C09105=1126.516,313.424,-77.649,-177.752,10.579,149.528
C09106=1126.520,313.176,-77.616,-177.755,10.576,149.528
C09107=1126.524,312.928,-77.584,-177.758,10.574,149.528
C09108=1126.528,312.680,-77.551,-177.761,10.571,149.528
C09109=1126.531,312.433,-77.519,-177.764,10.568,149.528
C09110=1126.536,312.184,-77.486,-177.767,10.567,149.529
C09111=1126.540,311.937,-77.453,-177.770,10.564,149.529
C09112=1126.544,311.688,-77.421,-177.773,10.562,149.529
C09113=1126.548,311.441,-77.389,-177.776,10.559,149.529
C09114=1126.552,311.193,-77.357,-177.779,10.556,149.529
C09115=1126.556,310.946,-77.324,-177.783,10.554,149.529
C09116=1126.560,310.698,-77.292,-177.786,10.551,149.530
C09117=1126.564,310.449,-77.259,-177.789,10.549,149.530
C09118=1126.568,310.202,-77.227,-177.792,10.546,149.530
C09119=1126.572,309.954,-77.194,-177.795,10.543,149.530
C09120=1126.577,309.706,-77.163,-177.798,10.541,149.530
C09121=1126.581,309.458,-77.130,-177.801,10.538,149.530
C09122=1126.584,309.210,-77.098,-177.805,10.536,149.531
C09123=1126.589,308.962,-77.065,-177.808,10.533,149.531
C09124=1126.592,308.715,-77.033,-177.811,10.531,149.531
C09125=1126.597,308.502,-77.005,-177.813,10.529,149.531
C09126=1126.600,308.289,-76.978,-177.816,10.527,149.531
C09127=1126.603,308.075,-76.950,-177.819,10.524,149.532
C09128=1126.607,307.862,-76.922,-177.821,10.522,149.532
C09129=1126.610,307.649,-76.895,-177.824,10.520,149.532
C09130=1126.614,307.436,-76.868,-177.827,10.518,149.532
C09131=1126.618,307.222,-76.840,-177.829,10.516,149.532
C09132=1126.621,307.009,-76.812,-177.832,10.513,149.532
C09133=1126.625,306.762,-76.779,-177.835,10.511,149.532
C09134=1126.629,306.514,-76.747,-177.838,10.509,149.533
C09135=1126.633,306.266,-76.715,-177.841,10.506,149.533
C09136=1126.637,306.017,-76.683,-177.844,10.504,149.533
C09137=1126.642,305.770,-76.652,-177.847,10.501,149.533
C09138=1126.645,305.522,-76.620,-177.851,10.499,149.533
C09139=1126.650,305.274,-76.587,-177.854,10.496,149.533
C09140=1126.653,305.026,-76.555,-177.857,10.493,149.534
C09141=1126.658,304.778,-76.524,-177.860,10.491,149.534
C09142=1126.662,304.530,-76.492,-177.863,10.488,149.534
C09143=1126.666,304.282,-76.460,-177.866,10.485,149.534
C09144=1126.670,304.035,-76.428,-177.869,10.483,149.534
C09145=1126.675,303.786,-76.396,-177.873,10.480,149.535
C09146=1126.678,303.538,-76.364,-177.876,10.478,149.535
C09147=1126.683,303.291,-76.332,-177.878,10.476,149.535
C09148=1126.687,303.043,-76.300,-177.881,10.473,149.535
C09149=1126.691,302.795,-76.268,-177.885,10.471,149.535
C09150=1126.695,302.547,-76.237,-177.888,10.468,149.536
C09151=1126.699,302.299,-76.205,-177.891,10.466,149.536
C09152=1126.703,302.051,-76.172,-177.894,10.463,149.536
C09153=1126.708,301.803,-76.141,-177.897,10.460,149.536
C09154=1126.711,301.555,-76.109,-177.900,10.458,149.536
C09155=1126.715,301.307,-76.077,-177.904,10.455,149.536
C09156=1126.720,301.059,-76.046,-177.906,10.452,149.537
C09157=1126.724,300.811,-76.014,-177.910,10.450,149.537
C09158=1126.728,300.563,-75.982,-177.913,10.447,149.537
C09159=1126.732,300.316,-75.951,-177.915,10.446,149.537
C09160=1126.736,300.068,-75.919,-177.918,10.443,149.537
C09161=1126.740,299.820,-75.888,-177.922,10.440,149.538
C09162=1126.745,299.571,-75.856,-177.925,10.438,149.538
C09163=1126.749,299.323,-75.824,-177.928,10.435,149.538
C09164=1126.753,299.076,-75.792,-177.931,10.432,149.538
C09165=1126.757,298.827,-75.761,-177.934,10.430,149.538
C09166=1126.761,298.579,-75.729,-177.937,10.427,149.538
C09167=1126.765,298.332,-75.698,-177.941,10.425,149.539
C09168=1126.769,298.084,-75.666,-177.943,10.422,149.539
C09169=1126.773,297.836,-75.635,-177.947,10.420,149.539
C09170=1126.777,297.588,-75.603,-177.950,10.417,149.539
C09171=1126.781,297.340,-75.573,-177.953,10.414,149.539
C09172=1126.785,297.092,-75.541,-177.955,10.412,149.539
C09173=1126.789,296.845,-75.509,-177.959,10.410,149.540
C09174=1126.794,296.596,-75.478,-177.962,10.407,149.540
C09175=1126.798,296.348,-75.446,-177.965,10.405,149.540
C09176=1126.803,296.100,-75.415,-177.968,10.402,149.540
C09177=1126.806,295.852,-75.383,-177.971,10.400,149.540
C09178=1126.811,295.604,-75.352,-177.974,10.397,149.540
C09179=1126.815,295.356,-75.321,-177.977,10.394,149.541
C09180=1126.818,295.109,-75.290,-177.980,10.392,149.541
C09181=1126.822,294.895,-75.263,-177.983,10.390,149.541
C09182=1126.826,294.682,-75.236,-177.985,10.388,149.541
C09183=1126.829,294.468,-75.209,-177.988,10.385,149.541
C09184=1126.833,294.255,-75.182,-177.991,10.383,149.541
C09185=1126.836,294.042,-75.155,-177.994,10.381,149.542
C09186=1126.840,293.828,-75.129,-177.996,10.379,149.542
C09187=1126.843,293.615,-75.101,-177.999,10.377,149.542
C09188=1126.847,293.401,-75.074,-178.002,10.374,149.542
C09189=1126.851,293.153,-75.044,-178.005,10.372,149.542
C09190=1126.855,292.905,-75.012,-178.008,10.369,149.543
C09191=1126.859,292.657,-74.981,-178.011,10.367,149.543
C09192=1126.864,292.409,-74.950,-178.013,10.365,149.543
C09193=1126.867,292.162,-74.919,-178.017,10.362,149.543
C09194=1126.872,291.914,-74.888,-178.020,10.359,149.543
C09195=1126.876,291.665,-74.857,-178.023,10.357,149.543
C09196=1126.880,291.418,-74.826,-178.026,10.354,149.544
C09197=1126.884,291.169,-74.795,-178.029,10.352,149.544
C09198=1126.889,290.921,-74.764,-178.032,10.349,149.544
C09199=1126.892,290.673,-74.733,-178.036,10.347,149.544
C09200=1126.896,290.426,-74.702,-178.039,10.344,149.544
C09201=1126.901,290.178,-74.671,-178.042,10.341,149.545
C09202=1126.905,289.929,-74.640,-178.044,10.339,149.545
C09203=1126.909,289.681,-74.609,-178.048,10.337,149.545
C09204=1126.912,289.433,-74.578,-178.050,10.334,149.545
C09205=1126.917,289.185,-74.547,-178.053,10.331,149.545
C09206=1126.922,288.937,-74.516,-178.057,10.329,149.545
C09207=1126.926,288.689,-74.485,-178.060,10.326,149.545
C09208=1126.929,288.441,-74.455,-178.063,10.324,149.546
C09209=1126.934,288.193,-74.424,-178.066,10.321,149.546
C09210=1126.938,287.945,-74.392,-178.069,10.319,149.546
C09211=1126.942,287.697,-74.362,-178.072,10.316,149.546
C09212=1126.946,287.449,-74.331,-178.075,10.314,149.546
C09213=1126.950,287.201,-74.300,-178.078,10.311,149.547
C09214=1126.955,286.953,-74.270,-178.081,10.309,149.547
C09215=1126.958,286.704,-74.239,-178.084,10.306,149.547
C09216=1126.963,286.456,-74.208,-178.087,10.304,149.547
C09217=1126.967,286.209,-74.178,-178.090,10.301,149.547
C09218=1126.971,285.960,-74.147,-178.093,10.298,149.547
C09219=1126.975,285.712,-74.116,-178.097,10.296,149.548
C09220=1126.980,285.464,-74.085,-178.100,10.293,149.548
C09221=1126.984,285.217,-74.055,-178.103,10.291,149.548
C09222=1126.988,284.968,-74.024,-178.105,10.289,149.548
C09223=1126.992,284.720,-73.993,-178.108,10.286,149.548
C09224=1126.996,284.472,-73.963,-178.112,10.284,149.549
C09225=1127.001,284.223,-73.933,-178.115,10.281,149.549
C09226=1127.004,283.975,-73.903,-178.118,10.278,149.549
C09227=1127.009,283.727,-73.872,-178.121,10.276,149.549
C09228=1127.013,283.480,-73.842,-178.124,10.273,149.549
C09229=1127.017,283.231,-73.811,-178.127,10.270,149.549
C09230=1127.022,282.983,-73.780,-178.130,10.268,149.549
C09231=1127.025,282.736,-73.750,-178.133,10.265,149.550
C09232=1127.030,282.487,-73.720,-178.136,10.263,149.550
C09233=1127.034,282.239,-73.689,-178.139,10.261,149.550
C09234=1127.038,281.991,-73.658,-178.142,10.258,149.550
C09235=1127.042,281.743,-73.628,-178.145,10.255,149.550
C09236=1127.047,281.494,-73.598,-178.148,10.253,149.551
C09237=1127.050,281.281,-73.572,-178.151,10.250,149.551
C09238=1127.054,281.068,-73.545,-178.154,10.248,149.551
C09239=1127.058,280.854,-73.520,-178.157,10.246,149.551
C09240=1127.061,280.641,-73.494,-178.160,10.243,149.551
C09241=1127.065,280.427,-73.468,-178.163,10.241,149.552
C09242=1127.068,280.214,-73.442,-178.166,10.238,149.552
C09243=1127.072,280.001,-73.415,-178.169,10.236,149.552
C09244=1127.075,279.787,-73.390,-178.172,10.234,149.552
C09245=1127.080,279.539,-73.359,-178.176,10.230,149.552
C09246=1127.084,279.291,-73.329,-178.179,10.228,149.553
C09247=1127.089,279.043,-73.299,-178.182,10.225,149.553
C09248=1127.093,278.795,-73.268,-178.185,10.223,149.553
C09249=1127.097,278.547,-73.239,-178.189,10.219,149.553
C09250=1127.101,278.298,-73.208,-178.192,10.217,149.553
C09251=1127.105,278.050,-73.178,-178.195,10.214,149.553
C09252=1127.109,277.802,-73.148,-178.198,10.212,149.554
C09253=1127.114,277.554,-73.118,-178.202,10.208,149.554
C09254=1127.118,277.306,-73.088,-178.205,10.206,149.554
C09255=1127.122,277.058,-73.059,-178.208,10.203,149.554
C09256=1127.126,276.810,-73.028,-178.211,10.200,149.554
C09257=1127.130,276.561,-72.998,-178.215,10.198,149.555
C09258=1127.134,276.313,-72.968,-178.218,10.194,149.555
C09259=1127.138,276.065,-72.938,-178.222,10.192,149.555
C09260=1127.143,275.816,-72.908,-178.224,10.189,149.555
C09261=1127.147,275.569,-72.878,-178.227,10.186,149.555
C09262=1127.151,275.320,-72.849,-178.230,10.183,149.555
C09263=1127.155,275.072,-72.819,-178.234,10.181,149.556
C09264=1127.160,274.824,-72.788,-178.237,10.178,149.556
C09265=1127.164,274.576,-72.759,-178.240,10.176,149.556
C09266=1127.168,274.328,-72.730,-178.243,10.173,149.556
C09267=1127.172,274.080,-72.699,-178.246,10.170,149.556
C09268=1127.177,273.831,-72.669,-178.249,10.168,149.556
C09269=1127.181,273.583,-72.640,-178.252,10.165,149.556
C09270=1127.185,273.335,-72.610,-178.255,10.162,149.556
C09271=1127.189,273.087,-72.580,-178.258,10.159,149.557
C09272=1127.193,272.839,-72.551,-178.261,10.157,149.557
C09273=1127.198,272.591,-72.521,-178.263,10.154,149.557
C09274=1127.202,272.342,-72.491,-178.267,10.151,149.557
C09275=1127.206,272.094,-72.461,-178.270,10.149,149.557
C09276=1127.210,271.846,-72.432,-178.273,10.146,149.557
C09277=1127.215,271.598,-72.402,-178.276,10.143,149.557
C09278=1127.219,271.350,-72.373,-178.278,10.141,149.557
C09279=1127.223,271.101,-72.343,-178.281,10.138,149.558
C09280=1127.227,270.853,-72.314,-178.284,10.136,149.558
C09281=1127.231,270.605,-72.284,-178.287,10.133,149.558
C09282=1127.235,270.357,-72.254,-178.290,10.130,149.558
C09283=1127.239,270.109,-72.225,-178.292,10.128,149.558
C09284=1127.244,269.860,-72.195,-178.295,10.125,149.558
C09285=1127.249,269.612,-72.165,-178.298,10.123,149.558
C09286=1127.253,269.364,-72.136,-178.300,10.121,149.558
C09287=1127.257,269.115,-72.106,-178.303,10.118,149.558
C09288=1127.261,268.867,-72.077,-178.306,10.115,149.558
C09289=1127.265,268.619,-72.047,-178.308,10.113,149.559
C09290=1127.269,268.371,-72.018,-178.311,10.110,149.559
C09291=1127.274,268.122,-71.989,-178.314,10.108,149.559
C09292=1127.278,267.874,-71.959,-178.317,10.106,149.559
C09293=1127.281,267.661,-71.934,-178.318,10.103,149.559
C09294=1127.285,267.447,-71.909,-178.321,10.101,149.559
C09295=1127.289,267.234,-71.884,-178.324,10.099,149.559
C09296=1127.292,267.020,-71.858,-178.326,10.097,149.559
C09297=1127.297,266.806,-71.833,-178.328,10.094,149.559
C09298=1127.300,266.593,-71.808,-178.330,10.092,149.559
C09299=1127.304,266.379,-71.783,-178.333,10.090,149.559
C09300=1127.307,266.166,-71.758,-178.335,10.088,149.560
C09301=1127.312,265.918,-71.728,-178.337,10.086,149.560
C09302=1127.316,265.669,-71.699,-178.339,10.084,149.560
C09303=1127.320,265.421,-71.669,-178.342,10.081,149.560
C09304=1127.324,265.173,-71.640,-178.344,10.079,149.560
C09305=1127.329,264.924,-71.611,-178.347,10.077,149.560
C09306=1127.333,264.676,-71.582,-178.350,10.075,149.560
C09307=1127.338,264.428,-71.553,-178.352,10.072,149.560
C09308=1127.341,264.180,-71.524,-178.356,10.069,149.560
C09309=1127.345,263.932,-71.494,-178.360,10.066,149.561
C09310=1127.350,263.683,-71.466,-178.363,10.063,149.561
C09311=1127.354,263.435,-71.436,-178.367,10.059,149.561
C09312=1127.359,263.187,-71.407,-178.371,10.056,149.561
C09313=1127.363,262.938,-71.378,-178.374,10.054,149.562
C09314=1127.367,262.690,-71.349,-178.378,10.050,149.562
C09315=1127.371,262.442,-71.320,-178.382,10.047,149.562
C09316=1127.375,262.193,-71.291,-178.385,10.044,149.562
C09317=1127.380,261.946,-71.262,-178.389,10.041,149.562
C09318=1127.384,261.697,-71.233,-178.392,10.038,149.563
C09319=1127.389,261.448,-71.204,-178.396,10.035,149.563
C09320=1127.392,261.200,-71.175,-178.400,10.032,149.563
C09321=1127.397,260.952,-71.146,-178.403,10.029,149.563
C09322=1127.401,260.704,-71.117,-178.406,10.025,149.563
C09323=1127.405,260.456,-71.089,-178.410,10.023,149.563
C09324=1127.409,260.207,-71.060,-178.413,10.020,149.564
C09325=1127.414,259.960,-71.031,-178.416,10.017,149.564
C09326=1127.419,259.711,-71.002,-178.419,10.014,149.564
C09327=1127.422,259.463,-70.973,-178.423,10.011,149.564
C09328=1127.427,259.214,-70.944,-178.426,10.008,149.564
C09329=1127.432,258.966,-70.916,-178.429,10.005,149.564
C09330=1127.435,258.718,-70.887,-178.433,10.002,149.564
C09331=1127.440,258.469,-70.858,-178.435,9.999,149.564
C09332=1127.444,258.221,-70.829,-178.438,9.996,149.565
C09333=1127.448,257.973,-70.801,-178.441,9.994,149.565
C09334=1127.453,257.724,-70.772,-178.444,9.991,149.565
C09335=1127.456,257.476,-70.744,-178.448,9.987,149.565
C09336=1127.461,257.228,-70.715,-178.451,9.985,149.565
C09337=1127.466,256.979,-70.686,-178.454,9.982,149.565
C09338=1127.470,256.731,-70.658,-178.456,9.979,149.565
C09339=1127.474,256.483,-70.629,-178.459,9.976,149.565
C09340=1127.478,256.234,-70.601,-178.462,9.973,149.565
C09341=1127.483,255.986,-70.572,-178.465,9.970,149.565
C09342=1127.486,255.738,-70.544,-178.465,9.969,149.565
C09343=1127.491,255.489,-70.515,-178.464,9.969,149.565
C09344=1127.496,255.241,-70.487,-178.465,9.967,149.565
C09345=1127.499,254.993,-70.458,-178.464,9.966,149.564
C09346=1127.504,254.744,-70.429,-178.465,9.965,149.564
C09347=1127.508,254.496,-70.401,-178.465,9.964,149.564
C09348=1127.513,254.247,-70.373,-178.466,9.963,149.564
C09349=1127.516,254.034,-70.347,-178.467,9.961,149.564
C09350=1127.519,253.820,-70.324,-178.468,9.960,149.564
C09351=1127.523,253.606,-70.299,-178.470,9.959,149.564
C09352=1127.528,253.393,-70.274,-178.471,9.957,149.564
C09353=1127.531,253.179,-70.250,-178.472,9.955,149.564
C09354=1127.535,252.965,-70.226,-178.474,9.954,149.564
C09355=1127.538,252.752,-70.201,-178.476,9.952,149.564
C09356=1127.542,252.538,-70.176,-178.478,9.950,149.564
C09357=1127.546,252.290,-70.149,-178.480,9.948,149.564
C09358=1127.551,252.041,-70.120,-178.484,9.946,149.564
C09359=1127.555,251.793,-70.092,-178.487,9.943,149.564
C09360=1127.559,251.545,-70.063,-178.490,9.940,149.565
C09361=1127.563,251.297,-70.034,-178.494,9.937,149.565
C09362=1127.568,251.048,-70.006,-178.498,9.934,149.565
C09363=1127.572,250.800,-69.978,-178.502,9.931,149.565
C09364=1127.576,250.551,-69.949,-178.506,9.928,149.566
C09365=1127.581,250.303,-69.921,-178.510,9.925,149.566
C09366=1127.584,250.054,-69.893,-178.515,9.921,149.566
C09367=1127.590,249.806,-69.865,-178.520,9.917,149.567
C09368=1127.593,249.558,-69.837,-178.525,9.913,149.567
C09369=1127.598,249.309,-69.808,-178.530,9.909,149.568
C09370=1127.602,249.061,-69.780,-178.536,9.904,149.568
C09371=1127.607,248.813,-69.752,-178.541,9.900,149.569
C09372=1127.611,248.564,-69.724,-178.548,9.895,149.569
C09373=1127.615,248.316,-69.696,-178.554,9.891,149.570
C09374=1127.619,248.068,-69.668,-178.560,9.886,149.570
C09375=1127.624,247.819,-69.641,-178.567,9.880,149.571
C09376=1127.628,247.570,-69.612,-178.574,9.875,149.571
C09377=1127.633,247.322,-69.584,-178.578,9.871,149.571
C09378=1127.637,247.075,-69.556,-178.580,9.868,149.571
C09379=1127.641,246.825,-69.529,-178.581,9.866,149.571
C09380=1127.646,246.577,-69.501,-178.583,9.864,149.571
C09381=1127.650,246.329,-69.472,-178.583,9.862,149.571
C09382=1127.655,246.080,-69.445,-178.585,9.860,149.571
C09383=1127.658,245.832,-69.417,-178.586,9.858,149.570
C09384=1127.663,245.584,-69.390,-178.588,9.856,149.570
C09385=1127.667,245.336,-69.362,-178.590,9.853,149.570
C09386=1127.672,245.086,-69.334,-178.591,9.851,149.570
C09387=1127.676,244.838,-69.306,-178.593,9.849,149.570
C09388=1127.680,244.590,-69.278,-178.595,9.847,149.570
C09389=1127.685,244.341,-69.251,-178.596,9.845,149.570
C09390=1127.689,244.093,-69.223,-178.598,9.843,149.570
C09391=1127.693,243.844,-69.196,-178.600,9.840,149.570
C09392=1127.698,243.596,-69.167,-178.602,9.838,149.570
C09393=1127.702,243.347,-69.139,-178.603,9.836,149.570
C09394=1127.706,243.099,-69.112,-178.605,9.833,149.570
C09395=1127.711,242.851,-69.084,-178.607,9.831,149.569
C09396=1127.715,242.603,-69.056,-178.609,9.829,149.569
C09397=1127.719,242.354,-69.029,-178.611,9.826,149.569
C09398=1127.724,242.106,-69.001,-178.613,9.824,149.569
C09399=1127.728,241.857,-68.974,-178.615,9.822,149.569
C09400=1127.732,241.609,-68.946,-178.617,9.820,149.569
C09401=1127.737,241.361,-68.919,-178.619,9.818,149.569
C09402=1127.741,241.112,-68.890,-178.621,9.815,149.569
C09403=1127.746,240.863,-68.863,-178.623,9.813,149.569
C09404=1127.750,240.615,-68.835,-178.626,9.810,149.569
C09405=1127.754,240.401,-68.812,-178.628,9.808,149.569
C09406=1127.757,240.187,-68.788,-178.629,9.807,149.569
C09407=1127.761,239.974,-68.764,-178.631,9.804,149.569
C09408=1127.765,239.760,-68.741,-178.634,9.802,149.570
C09409=1127.768,239.546,-68.717,-178.635,9.800,149.569
C09410=1127.772,239.332,-68.693,-178.638,9.798,149.570
C09411=1127.776,239.118,-68.670,-178.640,9.796,149.570
C09412=1127.780,238.905,-68.646,-178.642,9.794,149.570
C09413=1127.784,238.656,-68.618,-178.645,9.791,149.570
C09414=1127.788,238.408,-68.591,-178.647,9.789,149.570
C09415=1127.793,238.159,-68.564,-178.650,9.786,149.570
C09416=1127.797,237.910,-68.536,-178.652,9.784,149.570
C09417=1127.802,237.662,-68.508,-178.655,9.781,149.570
C09418=1127.806,237.414,-68.481,-178.658,9.778,149.570
C09419=1127.810,237.165,-68.455,-178.660,9.776,149.570
C09420=1127.814,236.917,-68.427,-178.663,9.773,149.570
C09421=1127.819,236.668,-68.400,-178.666,9.771,149.570
C09422=1127.823,236.420,-68.373,-178.669,9.768,149.571
C09423=1127.828,236.172,-68.345,-178.672,9.765,149.571
C09424=1127.832,235.923,-68.317,-178.675,9.762,149.571
C09425=1127.836,235.674,-68.290,-178.677,9.759,149.571
C09426=1127.841,235.426,-68.263,-178.680,9.756,149.571
C09427=1127.845,235.178,-68.235,-178.683,9.754,149.571
C09428=1127.849,234.929,-68.208,-178.686,9.751,149.571
C09429=1127.853,234.681,-68.182,-178.689,9.748,149.571
C09430=1127.858,234.432,-68.155,-178.692,9.745,149.571
C09431=1127.863,234.184,-68.127,-178.695,9.743,149.572
C09432=1127.867,233.936,-68.100,-178.698,9.740,149.572
C09433=1127.871,233.687,-68.072,-178.702,9.737,149.572
C09434=1127.876,233.438,-68.045,-178.705,9.734,149.572
C09435=1127.880,233.190,-68.019,-178.708,9.731,149.572
C09436=1127.884,232.941,-67.992,-178.711,9.728,149.572
C09437=1127.889,232.693,-67.965,-178.714,9.725,149.572
C09438=1127.893,232.444,-67.938,-178.718,9.722,149.573
C09439=1127.898,232.195,-67.910,-178.721,9.719,149.573
C09440=1127.901,231.947,-67.884,-178.724,9.715,149.573
C09441=1127.906,231.698,-67.857,-178.728,9.713,149.573
C09442=1127.911,231.450,-67.830,-178.731,9.709,149.573
C09443=1127.915,231.201,-67.802,-178.735,9.706,149.573
C09444=1127.919,230.953,-67.776,-178.738,9.703,149.573
C09445=1127.924,230.705,-67.749,-178.741,9.700,149.574
C09446=1127.929,230.456,-67.722,-178.745,9.696,149.574
C09447=1127.932,230.207,-67.695,-178.749,9.693,149.574
C09448=1127.937,229.959,-67.668,-178.753,9.689,149.574
C09449=1127.941,229.710,-67.641,-178.756,9.686,149.574
C09450=1127.945,229.462,-67.614,-178.760,9.682,149.574
C09451=1127.950,229.214,-67.587,-178.763,9.679,149.574
C09452=1127.955,228.965,-67.561,-178.767,9.676,149.575
C09453=1127.959,228.716,-67.535,-178.771,9.672,149.575
C09454=1127.963,228.468,-67.508,-178.774,9.669,149.575
C09455=1127.967,228.220,-67.481,-178.777,9.666,149.575
C09456=1127.972,227.971,-67.454,-178.781,9.662,149.575
C09457=1127.977,227.722,-67.428,-178.784,9.658,149.575
C09458=1127.981,227.474,-67.401,-178.788,9.655,149.575
C09459=1127.986,227.225,-67.374,-178.791,9.651,149.575
C09460=1127.990,226.977,-67.348,-178.794,9.649,149.576
C09461=1127.993,226.762,-67.325,-178.797,9.646,149.575
C09462=1127.997,226.549,-67.302,-178.800,9.642,149.576
C09463=1128.001,226.335,-67.280,-178.803,9.639,149.576
C09464=1128.005,226.121,-67.256,-178.806,9.636,149.576
C09465=1128.009,225.907,-67.234,-178.809,9.633,149.576
C09466=1128.012,225.693,-67.211,-178.811,9.630,149.576
C09467=1128.016,225.479,-67.188,-178.814,9.628,149.576
C09468=1128.020,225.265,-67.165,-178.816,9.625,149.576
C09469=1128.025,225.017,-67.139,-178.820,9.622,149.576
C09470=1128.029,224.768,-67.112,-178.823,9.618,149.576
C09471=1128.033,224.519,-67.086,-178.826,9.615,149.576
C09472=1128.037,224.271,-67.060,-178.828,9.612,149.576
C09473=1128.042,224.022,-67.034,-178.832,9.608,149.576
C09474=1128.046,223.774,-67.007,-178.834,9.605,149.576
C09475=1128.051,223.525,-66.981,-178.838,9.601,149.576
C09476=1128.055,223.276,-66.954,-178.840,9.598,149.576
C09477=1128.059,223.028,-66.929,-178.843,9.595,149.576
C09478=1128.064,222.779,-66.901,-178.846,9.592,149.576
C09479=1128.069,222.531,-66.876,-178.849,9.589,149.576
C09480=1128.073,222.283,-66.849,-178.851,9.586,149.576
C09481=1128.078,222.034,-66.823,-178.855,9.582,149.576
C09482=1128.082,221.785,-66.798,-178.857,9.579,149.576
C09483=1128.087,221.536,-66.770,-178.860,9.575,149.576
C09484=1128.091,221.288,-66.745,-178.862,9.572,149.576
C09485=1128.095,221.039,-66.718,-178.865,9.569,149.575
C09486=1128.099,220.791,-66.692,-178.867,9.566,149.575
C09487=1128.104,220.542,-66.667,-178.870,9.563,149.575
C09488=1128.108,220.294,-66.640,-178.872,9.560,149.575
C09489=1128.113,220.045,-66.614,-178.875,9.557,149.575
C09490=1128.118,219.796,-66.588,-178.877,9.554,149.575
C09491=1128.122,219.547,-66.562,-178.880,9.551,149.575
C09492=1128.126,219.299,-66.536,-178.882,9.547,149.575
C09493=1128.131,219.051,-66.510,-178.885,9.544,149.575
C09494=1128.136,218.802,-66.484,-178.887,9.541,149.575
C09495=1128.140,218.553,-66.458,-178.889,9.538,149.575
C09496=1128.144,218.305,-66.432,-178.892,9.535,149.575
C09497=1128.148,218.056,-66.406,-178.894,9.532,149.575
C09498=1128.152,217.807,-66.380,-178.896,9.529,149.574
C09499=1128.158,217.559,-66.354,-178.899,9.526,149.574
C09500=1128.162,217.310,-66.329,-178.900,9.523,149.574
C09501=1128.166,217.061,-66.303,-178.903,9.520,149.574
C09502=1128.170,216.813,-66.276,-178.905,9.517,149.574
C09503=1128.175,216.565,-66.251,-178.907,9.514,149.574
C09504=1128.179,216.316,-66.225,-178.909,9.511,149.574
C09505=1128.184,216.067,-66.199,-178.911,9.509,149.573
C09506=1128.188,215.818,-66.173,-178.913,9.506,149.573
C09507=1128.193,215.569,-66.147,-178.915,9.503,149.573
C09508=1128.197,215.321,-66.122,-178.917,9.500,149.573
C09509=1128.202,215.073,-66.096,-178.919,9.497,149.573
C09510=1128.206,214.824,-66.070,-178.921,9.494,149.573
C09511=1128.210,214.575,-66.045,-178.923,9.491,149.573
C09512=1128.215,214.327,-66.019,-178.925,9.489,149.573
C09513=1128.219,214.078,-65.994,-178.927,9.487,149.572
C09514=1128.224,213.829,-65.967,-178.929,9.483,149.572
C09515=1128.229,213.581,-65.942,-178.931,9.481,149.572
C09516=1128.233,213.332,-65.916,-178.932,9.478,149.572
C09517=1128.236,213.119,-65.894,-178.934,9.475,149.572
C09518=1128.240,212.904,-65.871,-178.935,9.474,149.572
C09519=1128.244,212.690,-65.850,-178.937,9.472,149.572
C09520=1128.248,212.475,-65.828,-178.938,9.470,149.571
C09521=1128.251,212.262,-65.806,-178.940,9.467,149.571
C09522=1128.256,212.048,-65.784,-178.941,9.465,149.571
C09523=1128.260,211.834,-65.762,-178.942,9.463,149.571
C09524=1128.263,211.620,-65.739,-178.944,9.461,149.571
C09525=1128.268,211.371,-65.714,-178.946,9.458,149.571
C09526=1128.272,211.122,-65.689,-178.949,9.455,149.571
C09527=1128.277,210.874,-65.663,-178.950,9.453,149.571
C09528=1128.281,210.625,-65.637,-178.952,9.450,149.571
C09529=1128.285,210.376,-65.612,-178.954,9.448,149.571
C09530=1128.290,210.128,-65.586,-178.956,9.445,149.571
C09531=1128.294,209.879,-65.561,-178.958,9.442,149.570
C09532=1128.299,209.631,-65.535,-178.961,9.440,149.571
C09533=1128.304,209.382,-65.510,-178.963,9.437,149.571
C09534=1128.308,209.133,-65.484,-178.966,9.434,149.571
C09535=1128.312,208.884,-65.459,-178.968,9.432,149.570
C09536=1128.317,208.636,-65.433,-178.970,9.429,149.570
C09537=1128.322,208.387,-65.408,-178.972,9.427,149.571
C09538=1128.326,208.138,-65.382,-178.975,9.424,149.571
C09539=1128.331,207.890,-65.357,-178.977,9.421,149.570
C09540=1128.335,207.641,-65.331,-178.980,9.419,149.571
C09541=1128.339,207.393,-65.307,-178.982,9.416,149.571
C09542=1128.344,207.144,-65.282,-178.985,9.414,149.571
C09543=1128.348,206.895,-65.256,-178.987,9.410,149.571
C09544=1128.353,206.647,-65.230,-178.990,9.408,149.571
C09545=1128.357,206.397,-65.205,-178.993,9.405,149.571
C09546=1128.362,206.149,-65.180,-178.996,9.402,149.571
C09547=1128.366,205.901,-65.154,-178.999,9.399,149.571
C09548=1128.371,205.651,-65.129,-179.001,9.396,149.571
C09549=1128.375,205.403,-65.104,-179.004,9.393,149.571
C09550=1128.379,205.154,-65.079,-179.007,9.391,149.571
C09551=1128.384,204.906,-65.054,-179.009,9.387,149.571
C09552=1128.388,204.657,-65.028,-179.012,9.385,149.571
C09553=1128.393,204.408,-65.004,-179.015,9.382,149.572
C09554=1128.398,204.160,-64.978,-179.018,9.379,149.572
C09555=1128.402,203.911,-64.954,-179.021,9.377,149.572
C09556=1128.406,203.662,-64.928,-179.024,9.373,149.572
C09557=1128.411,203.414,-64.903,-179.027,9.370,149.572
C09558=1128.416,203.165,-64.878,-179.030,9.367,149.572
C09559=1128.420,202.916,-64.853,-179.033,9.364,149.572
C09560=1128.424,202.668,-64.828,-179.037,9.361,149.572
C09561=1128.429,202.419,-64.803,-179.040,9.358,149.573
C09562=1128.433,202.170,-64.778,-179.043,9.355,149.573
C09563=1128.438,201.922,-64.753,-179.046,9.352,149.573
C09564=1128.443,201.672,-64.728,-179.050,9.348,149.573
C09565=1128.447,201.424,-64.703,-179.053,9.346,149.573
C09566=1128.451,201.175,-64.678,-179.057,9.342,149.573
C09567=1128.456,200.927,-64.653,-179.060,9.339,149.573
C09568=1128.460,200.678,-64.629,-179.064,9.335,149.573
C09569=1128.465,200.429,-64.604,-179.067,9.332,149.574
C09570=1128.469,200.180,-64.578,-179.070,9.329,149.574
C09571=1128.474,199.932,-64.554,-179.074,9.325,149.574
C09572=1128.478,199.682,-64.529,-179.077,9.322,149.574
C09573=1128.482,199.469,-64.508,-179.080,9.319,149.574
C09574=1128.486,199.255,-64.487,-179.083,9.316,149.574
C09575=1128.490,199.041,-64.466,-179.087,9.313,149.574
C09576=1128.494,198.826,-64.444,-179.090,9.310,149.575
C09577=1128.498,198.612,-64.423,-179.092,9.307,149.575
C09578=1128.502,198.398,-64.401,-179.096,9.303,149.575
C09579=1128.505,198.184,-64.380,-179.099,9.301,149.575
C09580=1128.509,197.969,-64.359,-179.102,9.297,149.575
C09581=1128.514,197.720,-64.334,-179.106,9.294,149.575
C09582=1128.518,197.471,-64.310,-179.110,9.290,149.575
C09583=1128.523,197.223,-64.285,-179.114,9.286,149.575
C09584=1128.527,196.975,-64.261,-179.117,9.282,149.576
C09585=1128.532,196.725,-64.235,-179.122,9.278,149.576
C09586=1128.536,196.477,-64.211,-179.125,9.275,149.576
C09587=1128.541,196.229,-64.187,-179.129,9.271,149.576
C09588=1128.545,195.979,-64.162,-179.130,9.268,149.576
C09589=1128.550,195.731,-64.138,-179.132,9.266,149.576
C09590=1128.555,195.482,-64.114,-179.134,9.263,149.575
C09591=1128.559,195.233,-64.089,-179.135,9.261,149.575
C09592=1128.564,194.984,-64.064,-179.137,9.258,149.575
C09593=1128.568,194.736,-64.040,-179.139,9.256,149.575
C09594=1128.572,194.487,-64.016,-179.140,9.253,149.575
C09595=1128.577,194.238,-63.991,-179.142,9.251,149.575
C09596=1128.581,193.990,-63.967,-179.143,9.248,149.574
C09597=1128.587,193.740,-63.943,-179.145,9.246,149.574
C09598=1128.591,193.491,-63.919,-179.147,9.243,149.574
C09599=1128.595,193.243,-63.895,-179.149,9.240,149.574
C09600=1128.600,192.994,-63.870,-179.150,9.238,149.574
C09601=1128.605,192.746,-63.846,-179.152,9.235,149.574
C09602=1128.608,192.496,-63.822,-179.154,9.233,149.574
C09603=1128.613,192.248,-63.797,-179.156,9.230,149.574
C09604=1128.618,191.999,-63.773,-179.158,9.227,149.574
C09605=1128.622,191.751,-63.749,-179.160,9.225,149.574
C09606=1128.627,191.501,-63.724,-179.161,9.222,149.573
C09607=1128.631,191.252,-63.700,-179.164,9.219,149.573
C09608=1128.636,191.004,-63.676,-179.166,9.217,149.573
C09609=1128.641,190.755,-63.652,-179.168,9.215,149.573
C09610=1128.645,190.506,-63.627,-179.170,9.211,149.573
C09611=1128.649,190.257,-63.604,-179.172,9.209,149.573
C09612=1128.655,190.008,-63.579,-179.173,9.206,149.573
C09613=1128.659,189.760,-63.555,-179.176,9.203,149.573
C09614=1128.663,189.512,-63.531,-179.178,9.201,149.573
C09615=1128.667,189.262,-63.507,-179.180,9.198,149.573
C09616=1128.673,189.013,-63.483,-179.182,9.196,149.573
C09617=1128.677,188.765,-63.458,-179.185,9.192,149.573
C09618=1128.681,188.516,-63.434,-179.187,9.190,149.573
C09619=1128.686,188.267,-63.411,-179.189,9.187,149.573
C09620=1128.691,188.018,-63.386,-179.192,9.184,149.573
C09621=1128.695,187.769,-63.362,-179.194,9.182,149.572
C09622=1128.700,187.520,-63.339,-179.196,9.178,149.572
C09623=1128.704,187.272,-63.315,-179.199,9.175,149.572
C09624=1128.709,187.024,-63.290,-179.201,9.173,149.572
C09625=1128.714,186.774,-63.266,-179.203,9.170,149.572
C09626=1128.718,186.525,-63.242,-179.206,9.167,149.572
C09627=1128.722,186.277,-63.218,-179.209,9.164,149.572
C09628=1128.727,186.028,-63.195,-179.211,9.161,149.572
C09629=1128.731,185.813,-63.174,-179.213,9.159,149.572
C09630=1128.735,185.599,-63.153,-179.215,9.156,149.572
C09631=1128.739,185.385,-63.133,-179.217,9.153,149.572
C09632=1128.742,185.170,-63.113,-179.219,9.151,149.572
C09633=1128.747,184.956,-63.092,-179.222,9.148,149.572
C09634=1128.751,184.742,-63.071,-179.224,9.146,149.572
C09635=1128.755,184.527,-63.051,-179.226,9.143,149.572
C09636=1128.758,184.313,-63.030,-179.229,9.140,149.572
C09637=1128.762,184.065,-63.006,-179.231,9.137,149.572
C09638=1128.768,183.815,-62.982,-179.234,9.134,149.572
C09639=1128.772,183.567,-62.958,-179.237,9.131,149.572
C09640=1128.777,183.318,-62.935,-179.239,9.128,149.572
C09641=1128.781,183.069,-62.911,-179.242,9.124,149.572
C09642=1128.786,182.820,-62.888,-179.245,9.122,149.572
C09643=1128.791,182.571,-62.864,-179.248,9.119,149.572
C09644=1128.795,182.323,-62.840,-179.250,9.115,149.572
C09645=1128.800,182.074,-62.817,-179.253,9.112,149.572
C09646=1128.804,181.826,-62.793,-179.256,9.109,149.572
C09647=1128.809,181.576,-62.769,-179.259,9.106,149.572
C09648=1128.814,181.327,-62.746,-179.262,9.102,149.572
C09649=1128.818,181.079,-62.722,-179.265,9.099,149.573
C09650=1128.823,180.830,-62.699,-179.268,9.095,149.573
C09651=1128.827,180.581,-62.675,-179.271,9.092,149.572
C09652=1128.832,180.332,-62.652,-179.274,9.089,149.573
C09653=1128.836,180.084,-62.628,-179.277,9.085,149.573
C09654=1128.840,179.835,-62.605,-179.280,9.082,149.573
C09655=1128.845,179.586,-62.582,-179.283,9.079,149.573
C09656=1128.850,179.337,-62.558,-179.286,9.075,149.573
C09657=1128.854,179.088,-62.534,-179.289,9.072,149.573
C09658=1128.859,178.839,-62.511,-179.291,9.069,149.573
C09659=1128.864,178.590,-62.487,-179.293,9.066,149.572
C09660=1128.868,178.341,-62.464,-179.295,9.063,149.572
C09661=1128.873,178.092,-62.441,-179.298,9.060,149.572
C09662=1128.877,177.843,-62.418,-179.299,9.057,149.572
C09663=1128.881,177.595,-62.394,-179.302,9.054,149.572
C09664=1128.886,177.346,-62.371,-179.304,9.052,149.572
C09665=1128.891,177.097,-62.347,-179.306,9.048,149.572
C09666=1128.895,176.848,-62.324,-179.308,9.045,149.572
C09667=1128.900,176.599,-62.300,-179.310,9.043,149.572
C09668=1128.904,176.350,-62.278,-179.312,9.039,149.571
C09669=1128.909,176.101,-62.254,-179.315,9.036,149.571
C09670=1128.913,175.852,-62.231,-179.317,9.034,149.571
C09671=1128.918,175.603,-62.208,-179.319,9.030,149.571
C09672=1128.923,175.355,-62.185,-179.321,9.027,149.571
C09673=1128.927,175.106,-62.162,-179.323,9.025,149.571
C09674=1128.932,174.857,-62.139,-179.325,9.021,149.571
C09675=1128.937,174.608,-62.115,-179.328,9.018,149.571
C09676=1128.942,174.359,-62.092,-179.330,9.016,149.571
C09677=1128.946,174.110,-62.069,-179.332,9.013,149.570
C09678=1128.950,173.861,-62.046,-179.334,9.009,149.570
C09679=1128.955,173.612,-62.022,-179.337,9.006,149.570
C09680=1128.960,173.364,-61.999,-179.339,9.004,149.570
C09681=1128.964,173.115,-61.977,-179.341,9.001,149.570
C09682=1128.969,172.866,-61.953,-179.343,8.997,149.570
C09683=1128.974,172.617,-61.930,-179.346,8.994,149.570
C09684=1128.978,172.368,-61.907,-179.348,8.992,149.570
C09685=1128.982,172.154,-61.887,-179.350,8.988,149.570
C09686=1128.986,171.939,-61.868,-179.352,8.986,149.570
C09687=1128.990,171.725,-61.848,-179.353,8.984,149.570
C09688=1128.994,171.510,-61.828,-179.355,8.982,149.570
C09689=1128.998,171.297,-61.808,-179.357,8.978,149.569
C09690=1129.002,171.081,-61.788,-179.359,8.976,149.569
C09691=1129.006,170.867,-61.769,-179.361,8.973,149.569
C09692=1129.010,170.653,-61.748,-179.363,8.971,149.569
C09693=1129.014,170.404,-61.726,-179.366,8.968,149.569
C09694=1129.019,170.155,-61.703,-179.368,8.964,149.569
C09695=1129.023,169.906,-61.681,-179.370,8.961,149.569
C09696=1129.028,169.657,-61.657,-179.373,8.958,149.569
C09697=1129.033,169.408,-61.634,-179.375,8.955,149.569
C09698=1129.037,169.159,-61.612,-179.377,8.952,149.569
C09699=1129.042,168.910,-61.589,-179.379,8.949,149.569
C09700=1129.046,168.662,-61.566,-179.382,8.946,149.569
C09701=1129.051,168.412,-61.543,-179.384,8.943,149.569
C09702=1129.055,168.163,-61.521,-179.386,8.940,149.568
C09703=1129.061,167.915,-61.498,-179.389,8.937,149.568
C09704=1129.066,167.665,-61.475,-179.392,8.933,149.568
C09705=1129.070,167.417,-61.452,-179.394,8.930,149.568
C09706=1129.075,167.168,-61.429,-179.396,8.927,149.568
C09707=1129.079,166.919,-61.407,-179.399,8.924,149.568
C09708=1129.084,166.670,-61.384,-179.401,8.921,149.568
C09709=1129.088,166.421,-61.362,-179.404,8.917,149.568
C09710=1129.093,166.172,-61.339,-179.406,8.914,149.568
C09711=1129.097,165.924,-61.316,-179.408,8.911,149.568
C09712=1129.102,165.674,-61.293,-179.411,8.908,149.568
C09713=1129.107,165.426,-61.271,-179.413,8.905,149.568
C09714=1129.111,165.177,-61.249,-179.415,8.901,149.567
C09715=1129.116,164.928,-61.226,-179.418,8.898,149.567
C09716=1129.121,164.679,-61.204,-179.420,8.895,149.567
C09717=1129.125,164.430,-61.181,-179.423,8.892,149.567
C09718=1129.130,164.181,-61.158,-179.425,8.888,149.567
C09719=1129.135,163.932,-61.136,-179.428,8.885,149.567
C09720=1129.139,163.683,-61.113,-179.430,8.882,149.567
C09721=1129.143,163.434,-61.091,-179.433,8.879,149.567
C09722=1129.149,163.185,-61.068,-179.435,8.876,149.567
C09723=1129.153,162.936,-61.046,-179.437,8.872,149.567
C09724=1129.157,162.687,-61.024,-179.440,8.869,149.567
C09725=1129.163,162.438,-61.001,-179.442,8.866,149.567
C09726=1129.167,162.189,-60.979,-179.444,8.863,149.566
C09727=1129.171,161.940,-60.957,-179.447,8.860,149.566
C09728=1129.177,161.691,-60.934,-179.449,8.857,149.566
C09729=1129.180,161.442,-60.911,-179.452,8.852,149.566
C09730=1129.185,161.194,-60.890,-179.455,8.849,149.566
C09731=1129.190,160.944,-60.867,-179.457,8.846,149.566
C09732=1129.195,160.695,-60.845,-179.460,8.843,149.566
C09733=1129.199,160.447,-60.823,-179.462,8.839,149.566
C09734=1129.203,160.197,-60.801,-179.464,8.836,149.566
C09735=1129.209,159.948,-60.778,-179.468,8.832,149.566
C09736=1129.213,159.699,-60.756,-179.470,8.829,149.566
C09737=1129.218,159.451,-60.734,-179.472,8.826,149.566
C09738=1129.222,159.202,-60.712,-179.475,8.823,149.565
C09739=1129.227,158.952,-60.689,-179.477,8.819,149.565
C09740=1129.232,158.704,-60.668,-179.480,8.815,149.565
C09741=1129.236,158.489,-60.648,-179.482,8.813,149.565
C09742=1129.240,158.274,-60.629,-179.484,8.810,149.565
C09743=1129.244,158.060,-60.610,-179.486,8.807,149.565
C09744=1129.248,157.845,-60.592,-179.488,8.804,149.565
C09745=1129.252,157.631,-60.572,-179.491,8.801,149.565
C09746=1129.256,157.416,-60.553,-179.493,8.798,149.565
C09747=1129.260,157.202,-60.534,-179.495,8.794,149.565
C09748=1129.264,156.987,-60.516,-179.497,8.792,149.565
C09749=1129.268,156.738,-60.494,-179.500,8.788,149.564
C09750=1129.273,156.489,-60.472,-179.503,8.785,149.564
C09751=1129.277,156.241,-60.449,-179.505,8.782,149.564
C09752=1129.282,155.992,-60.427,-179.508,8.777,149.564
C09753=1129.287,155.742,-60.405,-179.510,8.774,149.564
C09754=1129.292,155.494,-60.383,-179.513,8.771,149.564
C09755=1129.296,155.244,-60.361,-179.516,8.767,149.564
C09756=1129.301,154.996,-60.339,-179.518,8.764,149.564
C09757=1129.306,154.747,-60.318,-179.520,8.760,149.563
C09758=1129.311,154.497,-60.296,-179.523,8.756,149.563
C09759=1129.315,154.248,-60.275,-179.526,8.753,149.563
C09760=1129.320,153.999,-60.253,-179.529,8.749,149.563
C09761=1129.325,153.750,-60.231,-179.531,8.746,149.563
C09762=1129.329,153.501,-60.209,-179.534,8.742,149.563
C09763=1129.334,153.253,-60.187,-179.536,8.739,149.563
C09764=1129.339,153.004,-60.165,-179.539,8.734,149.563
C09765=1129.343,152.755,-60.143,-179.542,8.731,149.563
C09766=1129.348,152.506,-60.122,-179.544,8.727,149.562
C09767=1129.352,152.256,-60.100,-179.547,8.724,149.562
C09768=1129.357,152.007,-60.079,-179.549,8.720,149.562
C09769=1129.362,151.759,-60.057,-179.552,8.716,149.562
C09770=1129.366,151.509,-60.035,-179.555,8.712,149.562
C09771=1129.371,151.261,-60.013,-179.557,8.709,149.562
C09772=1129.376,151.011,-59.992,-179.560,8.705,149.562
C09773=1129.381,150.762,-59.970,-179.562,8.702,149.562
C09774=1129.385,150.513,-59.949,-179.565,8.697,149.561
C09775=1129.391,150.264,-59.928,-179.568,8.694,149.561
C09776=1129.395,150.015,-59.906,-179.570,8.690,149.561
C09777=1129.400,149.766,-59.884,-179.574,8.686,149.561
C09778=1129.404,149.517,-59.864,-179.576,8.682,149.561
C09779=1129.408,149.268,-59.842,-179.578,8.678,149.561
C09780=1129.413,149.019,-59.820,-179.582,8.675,149.561
C09781=1129.419,148.770,-59.799,-179.584,8.670,149.560
C09782=1129.423,148.521,-59.777,-179.587,8.667,149.560
C09783=1129.428,148.272,-59.755,-179.589,8.663,149.560
C09784=1129.432,148.023,-59.735,-179.592,8.659,149.560
C09785=1129.437,147.774,-59.713,-179.595,8.656,149.560
C09786=1129.442,147.524,-59.692,-179.597,8.651,149.560
C09787=1129.446,147.276,-59.670,-179.600,8.647,149.559
C09788=1129.452,147.027,-59.649,-179.603,8.643,149.559
C09789=1129.456,146.778,-59.628,-179.605,8.640,149.559
C09790=1129.460,146.528,-59.607,-179.608,8.635,149.559
C09791=1129.465,146.280,-59.585,-179.611,8.632,149.559
C09792=1129.470,146.030,-59.564,-179.614,8.627,149.559
C09793=1129.474,145.782,-59.543,-179.616,8.624,149.558
C09794=1129.479,145.532,-59.522,-179.619,8.619,149.558
C09795=1129.484,145.283,-59.501,-179.622,8.616,149.558
C09796=1129.488,145.034,-59.480,-179.625,8.611,149.558
C09797=1129.493,144.820,-59.461,-179.626,8.609,149.558
C09798=1129.497,144.605,-59.443,-179.627,8.606,149.557
C09799=1129.501,144.390,-59.425,-179.628,8.603,149.557
C09800=1129.505,144.176,-59.407,-179.629,8.600,149.557
C09801=1129.509,143.961,-59.389,-179.631,8.597,149.556
C09802=1129.513,143.746,-59.371,-179.632,8.594,149.556
C09803=1129.518,143.531,-59.352,-179.633,8.591,149.556
C09804=1129.521,143.317,-59.334,-179.634,8.588,149.555
C09805=1129.526,143.068,-59.313,-179.636,8.585,149.555
C09806=1129.531,142.819,-59.292,-179.637,8.582,149.555
C09807=1129.536,142.570,-59.271,-179.639,8.579,149.554
C09808=1129.540,142.321,-59.249,-179.640,8.576,149.554
C09809=1129.544,142.072,-59.229,-179.642,8.572,149.554
C09810=1129.550,141.823,-59.208,-179.643,8.569,149.553
C09811=1129.554,141.574,-59.188,-179.645,8.565,149.553
C09812=1129.559,141.325,-59.166,-179.646,8.563,149.553
C09813=1129.564,141.076,-59.145,-179.648,8.559,149.552
C09814=1129.569,140.827,-59.125,-179.649,8.556,149.552
C09815=1129.573,140.577,-59.103,-179.651,8.552,149.552
C09816=1129.577,140.328,-59.082,-179.652,8.549,149.551
C09817=1129.582,140.079,-59.061,-179.653,8.546,149.551
C09818=1129.587,139.830,-59.041,-179.655,8.542,149.550
C09819=1129.592,139.581,-59.020,-179.656,8.540,149.550
C09820=1129.596,139.332,-58.999,-179.658,8.536,149.550
C09821=1129.602,139.083,-58.978,-179.659,8.533,149.550
C09822=1129.606,138.834,-58.957,-179.661,8.529,149.549
C09823=1129.611,138.585,-58.936,-179.663,8.527,149.549
C09824=1129.615,138.336,-58.916,-179.664,8.523,149.548
C09825=1129.620,138.086,-58.895,-179.666,8.520,149.548
C09826=1129.624,137.837,-58.874,-179.667,8.516,149.548
C09827=1129.630,137.588,-58.853,-179.669,8.513,149.548
C09828=1129.634,137.339,-58.833,-179.670,8.510,149.547
C09829=1129.639,137.090,-58.812,-179.672,8.507,149.547
C09830=1129.644,136.841,-58.792,-179.673,8.503,149.546
C09831=1129.649,136.592,-58.771,-179.675,8.500,149.546
C09832=1129.653,136.343,-58.750,-179.677,8.497,149.546
C09833=1129.658,136.094,-58.729,-179.678,8.494,149.546
C09834=1129.663,135.845,-58.708,-179.680,8.490,149.545
C09835=1129.668,135.596,-58.687,-179.681,8.487,149.545
C09836=1129.672,135.347,-58.667,-179.683,8.484,149.545
C09837=1129.677,135.098,-58.647,-179.685,8.480,149.545
C09838=1129.682,134.849,-58.626,-179.686,8.477,149.544
C09839=1129.686,134.599,-58.606,-179.688,8.474,149.544
C09840=1129.692,134.350,-58.585,-179.689,8.470,149.543
C09841=1129.696,134.101,-58.565,-179.691,8.467,149.543
C09842=1129.701,133.852,-58.544,-179.693,8.464,149.543
C09843=1129.706,133.603,-58.523,-179.694,8.460,149.543
C09844=1129.710,133.354,-58.503,-179.696,8.458,149.542
C09845=1129.715,133.105,-58.482,-179.698,8.454,149.542
C09846=1129.720,132.856,-58.462,-179.700,8.450,149.542
C09847=1129.724,132.607,-58.441,-179.701,8.448,149.541
C09848=1129.729,132.357,-58.420,-179.703,8.444,149.541
C09849=1129.734,132.108,-58.400,-179.704,8.441,149.541
C09850=1129.739,131.859,-58.380,-179.706,8.437,149.541
C09851=1129.744,131.610,-58.359,-179.708,8.435,149.540
C09852=1129.748,131.361,-58.339,-179.709,8.431,149.540
C09853=1129.752,131.146,-58.321,-179.711,8.428,149.540
C09854=1129.757,130.931,-58.303,-179.712,8.425,149.539
C09855=1129.760,130.716,-58.286,-179.714,8.423,149.539
C09856=1129.765,130.502,-58.269,-179.715,8.420,149.539
C09857=1129.768,130.287,-58.251,-179.717,8.417,149.539
C09858=1129.773,130.072,-58.234,-179.718,8.413,149.538
C09859=1129.777,129.857,-58.216,-179.720,8.411,149.538
C09860=1129.780,129.643,-58.198,-179.721,8.408,149.538
C09861=1129.785,129.393,-58.178,-179.723,8.405,149.538
C09862=1129.791,129.145,-58.158,-179.725,8.402,149.537
C09863=1129.795,128.896,-58.137,-179.726,8.398,149.537
C09864=1129.800,128.646,-58.118,-179.728,8.395,149.537
C09865=1129.805,128.397,-58.097,-179.730,8.392,149.537
C09866=1129.810,128.148,-58.076,-179.732,8.388,149.536
C09867=1129.814,127.899,-58.056,-179.733,8.385,149.536
C09868=1129.819,127.649,-58.036,-179.735,8.382,149.536
C09869=1129.823,127.401,-58.016,-179.737,8.378,149.535
C09870=1129.828,127.152,-57.996,-179.738,8.375,149.535
C09871=1129.834,126.902,-57.976,-179.740,8.372,149.535
C09872=1129.838,126.653,-57.955,-179.742,8.368,149.535
C09873=1129.843,126.404,-57.936,-179.743,8.365,149.534
C09874=1129.847,126.155,-57.915,-179.746,8.362,149.534
C09875=1129.852,125.906,-57.895,-179.747,8.358,149.534
C09876=1129.857,125.656,-57.875,-179.749,8.355,149.534
C09877=1129.861,125.407,-57.855,-179.751,8.352,149.533
C09878=1129.867,125.158,-57.835,-179.753,8.348,149.533
C09879=1129.872,124.909,-57.815,-179.754,8.344,149.533
C09880=1129.876,124.660,-57.795,-179.756,8.342,149.532
C09881=1129.881,124.411,-57.775,-179.758,8.338,149.532
C09882=1129.886,124.161,-57.755,-179.760,8.335,149.532
C09883=1129.890,123.912,-57.735,-179.761,8.332,149.532
C09884=1129.895,123.663,-57.715,-179.763,8.328,149.531
C09885=1129.900,123.414,-57.695,-179.765,8.325,149.531
C09886=1129.904,123.165,-57.675,-179.767,8.321,149.531
C09887=1129.909,122.916,-57.655,-179.769,8.318,149.531
C09888=1129.914,122.666,-57.635,-179.771,8.315,149.530
C09889=1129.919,122.418,-57.615,-179.772,8.311,149.530
C09890=1129.923,122.169,-57.596,-179.774,8.308,149.530
C09891=1129.928,121.920,-57.575,-179.776,8.305,149.530
C09892=1129.933,121.670,-57.556,-179.778,8.301,149.529
C09893=1129.938,121.421,-57.536,-179.780,8.298,149.529
C09894=1129.942,121.172,-57.516,-179.782,8.294,149.529
C09895=1129.947,120.923,-57.496,-179.784,8.290,149.528
C09896=1129.952,120.674,-57.476,-179.785,8.288,149.528
C09897=1129.956,120.424,-57.456,-179.787,8.284,149.528
C09898=1129.962,120.175,-57.437,-179.789,8.281,149.528
C09899=1129.966,119.926,-57.417,-179.791,8.277,149.527
C09900=1129.971,119.677,-57.397,-179.793,8.273,149.527
C09901=1129.976,119.428,-57.378,-179.794,8.271,149.527
C09902=1129.981,119.178,-57.358,-179.796,8.267,149.527
C09903=1129.985,118.929,-57.338,-179.798,8.264,149.526
C09904=1129.990,118.680,-57.318,-179.801,8.260,149.526
C09905=1129.995,118.431,-57.299,-179.802,8.256,149.526
C09906=1130.000,118.182,-57.278,-179.804,8.253,149.526
C09907=1130.005,117.932,-57.259,-179.806,8.250,149.525
C09908=1130.010,117.684,-57.239,-179.808,8.247,149.525
C09909=1130.014,117.468,-57.222,-179.810,8.243,149.525
C09910=1130.018,117.253,-57.205,-179.811,8.240,149.525
C09911=1130.022,117.039,-57.188,-179.813,8.238,149.525
C09912=1130.026,116.824,-57.172,-179.815,8.234,149.524
C09913=1130.030,116.609,-57.155,-179.816,8.231,149.524
C09914=1130.034,116.395,-57.138,-179.818,8.229,149.524
C09915=1130.038,116.179,-57.121,-179.820,8.225,149.524
C09916=1130.043,115.965,-57.104,-179.821,8.222,149.523
C09917=1130.047,115.715,-57.085,-179.823,8.219,149.523
C09918=1130.052,115.466,-57.065,-179.825,8.215,149.523
C09919=1130.058,115.217,-57.046,-179.827,8.212,149.523
C09920=1130.062,114.968,-57.027,-179.829,8.208,149.522
C09921=1130.066,114.718,-57.007,-179.831,8.205,149.522
C09922=1130.071,114.470,-56.987,-179.833,8.201,149.522
C09923=1130.076,114.220,-56.968,-179.834,8.198,149.521
C09924=1130.081,113.971,-56.948,-179.836,8.195,149.521
C09925=1130.085,113.722,-56.929,-179.838,8.191,149.521
C09926=1130.090,113.473,-56.910,-179.840,8.188,149.521
C09927=1130.096,113.224,-56.890,-179.842,8.184,149.521
C09928=1130.100,112.974,-56.871,-179.844,8.180,149.520
C09929=1130.105,112.726,-56.852,-179.846,8.177,149.520
C09930=1130.110,112.476,-56.832,-179.848,8.173,149.520
C09931=1130.115,112.227,-56.813,-179.850,8.170,149.519
C09932=1130.120,111.978,-56.793,-179.852,8.166,149.519
C09933=1130.124,111.728,-56.774,-179.854,8.162,149.519
C09934=1130.129,111.479,-56.756,-179.856,8.159,149.519
C09935=1130.134,111.229,-56.736,-179.858,8.155,149.518
C09936=1130.139,110.981,-56.717,-179.860,8.152,149.518
C09937=1130.143,110.731,-56.698,-179.863,8.147,149.518
C09938=1130.149,110.482,-56.678,-179.865,8.144,149.518
C09939=1130.153,110.233,-56.659,-179.867,8.140,149.518
C09940=1130.158,109.984,-56.640,-179.870,8.135,149.517
C09941=1130.163,109.735,-56.620,-179.873,8.132,149.517
C09942=1130.168,109.486,-56.602,-179.875,8.128,149.517
C09943=1130.173,109.236,-56.583,-179.878,8.124,149.517
C09944=1130.178,108.987,-56.563,-179.880,8.120,149.517
C09945=1130.182,108.738,-56.544,-179.883,8.116,149.516
C09946=1130.187,108.489,-56.525,-179.885,8.112,149.516
C09947=1130.192,108.239,-56.507,-179.887,8.108,149.516
C09948=1130.197,107.990,-56.487,-179.890,8.104,149.516
C09949=1130.201,107.741,-56.468,-179.893,8.100,149.516
C09950=1130.207,107.491,-56.450,-179.895,8.096,149.515
C09951=1130.211,107.242,-56.430,-179.898,8.092,149.515
C09952=1130.216,106.993,-56.411,-179.900,8.088,149.515
C09953=1130.221,106.743,-56.392,-179.902,8.084,149.515
C09954=1130.226,106.495,-56.374,-179.905,8.080,149.514
C09955=1130.231,106.246,-56.354,-179.907,8.076,149.514
C09956=1130.235,105.996,-56.336,-179.910,8.072,149.514
C09957=1130.241,105.747,-56.317,-179.912,8.068,149.514
C09958=1130.245,105.498,-56.298,-179.914,8.064,149.513
C09959=1130.249,105.249,-56.280,-179.916,8.060,149.513
C09960=1130.254,104.999,-56.260,-179.919,8.056,149.513
C09961=1130.259,104.750,-56.242,-179.921,8.053,149.513
C09962=1130.264,104.501,-56.223,-179.924,8.048,149.512
C09963=1130.269,104.251,-56.205,-179.926,8.044,149.512
C09964=1130.274,104.002,-56.185,-179.928,8.040,149.512
C09965=1130.278,103.787,-56.170,-179.930,8.037,149.512
C09966=1130.282,103.572,-56.153,-179.932,8.033,149.511
C09967=1130.286,103.358,-56.137,-179.934,8.030,149.511
C09968=1130.291,103.142,-56.121,-179.936,8.026,149.511
C09969=1130.294,102.928,-56.105,-179.937,8.023,149.511
C09970=1130.299,102.713,-56.089,-179.939,8.019,149.510
C09971=1130.303,102.497,-56.073,-179.941,8.016,149.510
C09972=1130.307,102.283,-56.057,-179.943,8.012,149.510
C09973=1130.312,102.034,-56.039,-179.945,8.009,149.510
C09974=1130.317,101.784,-56.019,-179.947,8.004,149.509
C09975=1130.322,101.535,-56.001,-179.950,8.001,149.509
C09976=1130.327,101.286,-55.983,-179.952,7.996,149.509
C09977=1130.332,101.036,-55.963,-179.954,7.993,149.508
C09978=1130.336,100.787,-55.945,-179.955,7.989,149.508
C09979=1130.341,100.538,-55.927,-179.958,7.984,149.508
C09980=1130.345,100.289,-55.908,-179.960,7.981,149.507
C09981=1130.351,100.039,-55.890,-179.962,7.976,149.507
C09982=1130.356,99.790,-55.872,-179.964,7.972,149.507
C09983=1130.361,99.541,-55.853,-179.966,7.969,149.506
C09984=1130.365,99.291,-55.835,-179.968,7.964,149.506
C09985=1130.371,99.042,-55.816,-179.970,7.960,149.506
C09986=1130.375,98.793,-55.798,-179.972,7.957,149.505
C09987=1130.380,98.544,-55.780,-179.974,7.952,149.505
C09988=1130.384,98.294,-55.761,-179.976,7.949,149.505
C09989=1130.390,98.045,-55.743,-179.978,7.945,149.504
C09990=1130.395,97.796,-55.725,-179.980,7.940,149.504
C09991=1130.400,97.547,-55.707,-179.982,7.936,149.503
C09992=1130.404,97.297,-55.688,-179.984,7.933,149.503
C09993=1130.409,97.048,-55.670,-179.985,7.929,149.503
C09994=1130.414,96.799,-55.652,-179.988,7.924,149.502
C09995=1130.419,96.549,-55.633,-179.990,7.921,149.502
C09996=1130.424,96.300,-55.615,-179.991,7.917,149.502
//INST
///DATE 2021/06/25 14:32
///ATTR SC,RW,RJ
////FRAME ROBOT
///GROUP1 RB1
NOP
MOVL C00000 V=800.0 PL=0
MOVL C00001 V=800.0 PL=0
MOVL C00002 V=800.0 PL=0
MOVL C00003 V=800.0 PL=0
MOVL C00004 V=800.0 PL=0
MOVL C00005 V=800.0 PL=0
MOVL C00006 V=800.0 PL=0
MOVL C00007 V=800.0 PL=0
MOVL C00008 V=800.0 PL=0
MOVL C00009 V=800.0 PL=0
MOVL C00010 V=800.0 PL=0
MOVL C00011 V=800.0 PL=0
MOVL C00012 V=800.0 PL=0
MOVL C00013 V=800.0 PL=0
MOVL C00014 V=800.0 PL=0
MOVL C00015 V=800.0 PL=0
MOVL C00016 V=800.0 PL=0
MOVL C00017 V=800.0 PL=0
MOVL C00018 V=800.0 PL=0
MOVL C00019 V=800.0 PL=0
MOVL C00020 V=800.0 PL=0
MOVL C00021 V=800.0 PL=0
MOVL C00022 V=800.0 PL=0
MOVL C00023 V=800.0 PL=0
MOVL C00024 V=800.0 PL=0
MOVL C00025 V=800.0 PL=0
MOVL C00026 V=800.0 PL=0
MOVL C00027 V=800.0 PL=0
MOVL C00028 V=800.0 PL=0
MOVL C00029 V=800.0 PL=0
MOVL C00030 V=800.0 PL=0
MOVL C00031 V=800.0 PL=0
MOVL C00032 V=800.0 PL=0
MOVL C00033 V=800.0 PL=0
MOVL C00034 V=800.0 PL=0
MOVL C00035 V=800.0 PL=0
MOVL C00036 V=800.0 PL=0
MOVL C00037 V=800.0 PL=0
MOVL C00038 V=800.0 PL=0
MOVL C00039 V=800.0 PL=0
MOVL C00040 V=800.0 PL=0
MOVL C00041 V=800.0 PL=0
MOVL C00042 V=800.0 PL=0
MOVL C00043 V=800.0 PL=0
MOVL C00044 V=800.0 PL=0
MOVL C00045 V=800.0 PL=0
MOVL C00046 V=800.0 PL=0
MOVL C00047 V=800.0 PL=0
MOVL C00048 V=800.0 PL=0
MOVL C00049 V=800.0 PL=0
MOVL C00050 V=800.0 PL=0
MOVL C00051 V=800.0 PL=0
MOVL C00052 V=800.0 PL=0
MOVL C00053 V=800.0 PL=0
MOVL C00054 V=800.0 PL=0
MOVL C00055 V=800.0 PL=0
MOVL C00056 V=800.0 PL=0
MOVL C00057 V=800.0 PL=0
MOVL C00058 V=800.0 PL=0
MOVL C00059 V=800.0 PL=0
MOVL C00060 V=800.0 PL=0
MOVL C00061 V=800.0 PL=0
MOVL C00062 V=800.0 PL=0
MOVL C00063 V=800.0 PL=0
MOVL C00064 V=800.0 PL=0
MOVL C00065 V=800.0 PL=0
MOVL C00066 V=800.0 PL=0
MOVL C00067 V=800.0 PL=0
MOVL C00068 V=800.0 PL=0
MOVL C00069 V=800.0 PL=0
MOVL C00070 V=800.0 PL=0
MOVL C00071 V=800.0 PL=0
MOVL C00072 V=800.0 PL=0
MOVL C00073 V=800.0 PL=0
MOVL C00074 V=800.0 PL=0
MOVL C00075 V=800.0 PL=0
MOVL C00076 V=800.0 PL=0
MOVL C00077 V=800.0 PL=0
MOVL C00078 V=800.0 PL=0
MOVL C00079 V=800.0 PL=0
MOVL C00080 V=800.0 PL=0
MOVL C00081 V=800.0 PL=0
MOVL C00082 V=800.0 PL=0
MOVL C00083 V=800.0 PL=0
MOVL C00084 V=800.0 PL=0
MOVL C00085 V=800.0 PL=0
MOVL C00086 V=800.0 PL=0
MOVL C00087 V=800.0 PL=0
MOVL C00088 V=800.0 PL=0
MOVL C00089 V=800.0 PL=0
MOVL C00090 V=800.0 PL=0
MOVL C00091 V=800.0 PL=0
MOVL C00092 V=800.0 PL=0
MOVL C00093 V=800.0 PL=0
MOVL C00094 V=800.0 PL=0
MOVL C00095 V=800.0 PL=0
MOVL C00096 V=800.0 PL=0
MOVL C00097 V=800.0 PL=0
MOVL C00098 V=800.0 PL=0
MOVL C00099 V=800.0 PL=0
MOVL C00100 V=800.0 PL=0
MOVL C00101 V=800.0 PL=0
MOVL C00102 V=800.0 PL=0
MOVL C00103 V=800.0 PL=0
MOVL C00104 V=800.0 PL=0
MOVL C00105 V=800.0 PL=0
MOVL C00106 V=800.0 PL=0
MOVL C00107 V=800.0 PL=0
MOVL C00108 V=800.0 PL=0
MOVL C00109 V=800.0 PL=0
MOVL C00110 V=800.0 PL=0
MOVL C00111 V=800.0 PL=0
MOVL C00112 V=800.0 PL=0
MOVL C00113 V=800.0 PL=0
MOVL C00114 V=800.0 PL=0
MOVL C00115 V=800.0 PL=0
MOVL C00116 V=800.0 PL=0
MOVL C00117 V=800.0 PL=0
MOVL C00118 V=800.0 PL=0
MOVL C00119 V=800.0 PL=0
MOVL C00120 V=800.0 PL=0
MOVL C00121 V=800.0 PL=0
MOVL C00122 V=800.0 PL=0
MOVL C00123 V=800.0 PL=0
MOVL C00124 V=800.0 PL=0
MOVL C00125 V=800.0 PL=0
MOVL C00126 V=800.0 PL=0
MOVL C00127 V=800.0 PL=0
MOVL C00128 V=800.0 PL=0
MOVL C00129 V=800.0 PL=0
MOVL C00130 V=800.0 PL=0
MOVL C00131 V=800.0 PL=0
MOVL C00132 V=800.0 PL=0
MOVL C00133 V=800.0 PL=0
MOVL C00134 V=800.0 PL=0
MOVL C00135 V=800.0 PL=0
MOVL C00136 V=800.0 PL=0
MOVL C00137 V=800.0 PL=0
MOVL C00138 V=800.0 PL=0
MOVL C00139 V=800.0 PL=0
MOVL C00140 V=800.0 PL=0
MOVL C00141 V=800.0 PL=0
MOVL C00142 V=800.0 PL=0
MOVL C00143 V=800.0 PL=0
MOVL C00144 V=800.0 PL=0
MOVL C00145 V=800.0 PL=0
MOVL C00146 V=800.0 PL=0
MOVL C00147 V=800.0 PL=0
MOVL C00148 V=800.0 PL=0
MOVL C00149 V=800.0 PL=0
MOVL C00150 V=800.0 PL=0
MOVL C00151 V=800.0 PL=0
MOVL C00152 V=800.0 PL=0
MOVL C00153 V=800.0 PL=0
MOVL C00154 V=800.0 PL=0
MOVL C00155 V=800.0 PL=0
MOVL C00156 V=800.0 PL=0
MOVL C00157 V=800.0 PL=0
MOVL C00158 V=800.0 PL=0
MOVL C00159 V=800.0 PL=0
MOVL C00160 V=800.0 PL=0
MOVL C00161 V=800.0 PL=0
MOVL C00162 V=800.0 PL=0
MOVL C00163 V=800.0 PL=0
MOVL C00164 V=800.0 PL=0
MOVL C00165 V=800.0 PL=0
MOVL C00166 V=800.0 PL=0
MOVL C00167 V=800.0 PL=0
MOVL C00168 V=800.0 PL=0
MOVL C00169 V=800.0 PL=0
MOVL C00170 V=800.0 PL=0
MOVL C00171 V=800.0 PL=0
MOVL C00172 V=800.0 PL=0
MOVL C00173 V=800.0 PL=0
MOVL C00174 V=800.0 PL=0
MOVL C00175 V=800.0 PL=0
MOVL C00176 V=800.0 PL=0
MOVL C00177 V=800.0 PL=0
MOVL C00178 V=800.0 PL=0
MOVL C00179 V=800.0 PL=0
MOVL C00180 V=800.0 PL=0
MOVL C00181 V=800.0 PL=0
MOVL C00182 V=800.0 PL=0
MOVL C00183 V=800.0 PL=0
MOVL C00184 V=800.0 PL=0
MOVL C00185 V=800.0 PL=0
MOVL C00186 V=800.0 PL=0
MOVL C00187 V=800.0 PL=0
MOVL C00188 V=800.0 PL=0
MOVL C00189 V=800.0 PL=0
MOVL C00190 V=800.0 PL=0
MOVL C00191 V=800.0 PL=0
MOVL C00192 V=800.0 PL=0
MOVL C00193 V=800.0 PL=0
MOVL C00194 V=800.0 PL=0
MOVL C00195 V=800.0 PL=0
MOVL C00196 V=800.0 PL=0
MOVL C00197 V=800.0 PL=0
MOVL C00198 V=800.0 PL=0
MOVL C00199 V=800.0 PL=0
MOVL C00200 V=800.0 PL=0
MOVL C00201 V=800.0 PL=0
MOVL C00202 V=800.0 PL=0
MOVL C00203 V=800.0 PL=0
MOVL C00204 V=800.0 PL=0
MOVL C00205 V=800.0 PL=0
MOVL C00206 V=800.0 PL=0
MOVL C00207 V=800.0 PL=0
MOVL C00208 V=800.0 PL=0
MOVL C00209 V=800.0 PL=0
MOVL C00210 V=800.0 PL=0
MOVL C00211 V=800.0 PL=0
MOVL C00212 V=800.0 PL=0
MOVL C00213 V=800.0 PL=0
MOVL C00214 V=800.0 PL=0
MOVL C00215 V=800.0 PL=0
MOVL C00216 V=800.0 PL=0
MOVL C00217 V=800.0 PL=0
MOVL C00218 V=800.0 PL=0
MOVL C00219 V=800.0 PL=0
MOVL C00220 V=800.0 PL=0
MOVL C00221 V=800.0 PL=0
MOVL C00222 V=800.0 PL=0
MOVL C00223 V=800.0 PL=0
MOVL C00224 V=800.0 PL=0
MOVL C00225 V=800.0 PL=0
MOVL C00226 V=800.0 PL=0
MOVL C00227 V=800.0 PL=0
MOVL C00228 V=800.0 PL=0
MOVL C00229 V=800.0 PL=0
MOVL C00230 V=800.0 PL=0
MOVL C00231 V=800.0 PL=0
MOVL C00232 V=800.0 PL=0
MOVL C00233 V=800.0 PL=0
MOVL C00234 V=800.0 PL=0
MOVL C00235 V=800.0 PL=0
MOVL C00236 V=800.0 PL=0
MOVL C00237 V=800.0 PL=0
MOVL C00238 V=800.0 PL=0
MOVL C00239 V=800.0 PL=0
MOVL C00240 V=800.0 PL=0
MOVL C00241 V=800.0 PL=0
MOVL C00242 V=800.0 PL=0
MOVL C00243 V=800.0 PL=0
MOVL C00244 V=800.0 PL=0
MOVL C00245 V=800.0 PL=0
MOVL C00246 V=800.0 PL=0
MOVL C00247 V=800.0 PL=0
MOVL C00248 V=800.0 PL=0
MOVL C00249 V=800.0 PL=0
MOVL C00250 V=800.0 PL=0
MOVL C00251 V=800.0 PL=0
MOVL C00252 V=800.0 PL=0
MOVL C00253 V=800.0 PL=0
MOVL C00254 V=800.0 PL=0
MOVL C00255 V=800.0 PL=0
MOVL C00256 V=800.0 PL=0
MOVL C00257 V=800.0 PL=0
MOVL C00258 V=800.0 PL=0
MOVL C00259 V=800.0 PL=0
MOVL C00260 V=800.0 PL=0
MOVL C00261 V=800.0 PL=0
MOVL C00262 V=800.0 PL=0
MOVL C00263 V=800.0 PL=0
MOVL C00264 V=800.0 PL=0
MOVL C00265 V=800.0 PL=0
MOVL C00266 V=800.0 PL=0
MOVL C00267 V=800.0 PL=0
MOVL C00268 V=800.0 PL=0
MOVL C00269 V=800.0 PL=0
MOVL C00270 V=800.0 PL=0
MOVL C00271 V=800.0 PL=0
MOVL C00272 V=800.0 PL=0
MOVL C00273 V=800.0 PL=0
MOVL C00274 V=800.0 PL=0
MOVL C00275 V=800.0 PL=0
MOVL C00276 V=800.0 PL=0
MOVL C00277 V=800.0 PL=0
MOVL C00278 V=800.0 PL=0
MOVL C00279 V=800.0 PL=0
MOVL C00280 V=800.0 PL=0
MOVL C00281 V=800.0 PL=0
MOVL C00282 V=800.0 PL=0
MOVL C00283 V=800.0 PL=0
MOVL C00284 V=800.0 PL=0
MOVL C00285 V=800.0 PL=0
MOVL C00286 V=800.0 PL=0
MOVL C00287 V=800.0 PL=0
MOVL C00288 V=800.0 PL=0
MOVL C00289 V=800.0 PL=0
MOVL C00290 V=800.0 PL=0
MOVL C00291 V=800.0 PL=0
MOVL C00292 V=800.0 PL=0
MOVL C00293 V=800.0 PL=0
MOVL C00294 V=800.0 PL=0
MOVL C00295 V=800.0 PL=0
MOVL C00296 V=800.0 PL=0
MOVL C00297 V=800.0 PL=0
MOVL C00298 V=800.0 PL=0
MOVL C00299 V=800.0 PL=0
MOVL C00300 V=800.0 PL=0
MOVL C00301 V=800.0 PL=0
MOVL C00302 V=800.0 PL=0
MOVL C00303 V=800.0 PL=0
MOVL C00304 V=800.0 PL=0
MOVL C00305 V=800.0 PL=0
MOVL C00306 V=800.0 PL=0
MOVL C00307 V=800.0 PL=0
MOVL C00308 V=800.0 PL=0
MOVL C00309 V=800.0 PL=0
MOVL C00310 V=800.0 PL=0
MOVL C00311 V=800.0 PL=0
MOVL C00312 V=800.0 PL=0
MOVL C00313 V=800.0 PL=0
MOVL C00314 V=800.0 PL=0
MOVL C00315 V=800.0 PL=0
MOVL C00316 V=800.0 PL=0
MOVL C00317 V=800.0 PL=0
MOVL C00318 V=800.0 PL=0
MOVL C00319 V=800.0 PL=0
MOVL C00320 V=800.0 PL=0
MOVL C00321 V=800.0 PL=0
MOVL C00322 V=800.0 PL=0
MOVL C00323 V=800.0 PL=0
MOVL C00324 V=800.0 PL=0
MOVL C00325 V=800.0 PL=0
MOVL C00326 V=800.0 PL=0
MOVL C00327 V=800.0 PL=0
MOVL C00328 V=800.0 PL=0
MOVL C00329 V=800.0 PL=0
MOVL C00330 V=800.0 PL=0
MOVL C00331 V=800.0 PL=0
MOVL C00332 V=800.0 PL=0
MOVL C00333 V=800.0 PL=0
MOVL C00334 V=800.0 PL=0
MOVL C00335 V=800.0 PL=0
MOVL C00336 V=800.0 PL=0
MOVL C00337 V=800.0 PL=0
MOVL C00338 V=800.0 PL=0
MOVL C00339 V=800.0 PL=0
MOVL C00340 V=800.0 PL=0
MOVL C00341 V=800.0 PL=0
MOVL C00342 V=800.0 PL=0
MOVL C00343 V=800.0 PL=0
MOVL C00344 V=800.0 PL=0
MOVL C00345 V=800.0 PL=0
MOVL C00346 V=800.0 PL=0
MOVL C00347 V=800.0 PL=0
MOVL C00348 V=800.0 PL=0
MOVL C00349 V=800.0 PL=0
MOVL C00350 V=800.0 PL=0
MOVL C00351 V=800.0 PL=0
MOVL C00352 V=800.0 PL=0
MOVL C00353 V=800.0 PL=0
MOVL C00354 V=800.0 PL=0
MOVL C00355 V=800.0 PL=0
MOVL C00356 V=800.0 PL=0
MOVL C00357 V=800.0 PL=0
MOVL C00358 V=800.0 PL=0
MOVL C00359 V=800.0 PL=0
MOVL C00360 V=800.0 PL=0
MOVL C00361 V=800.0 PL=0
MOVL C00362 V=800.0 PL=0
MOVL C00363 V=800.0 PL=0
MOVL C00364 V=800.0 PL=0
MOVL C00365 V=800.0 PL=0
MOVL C00366 V=800.0 PL=0
MOVL C00367 V=800.0 PL=0
MOVL C00368 V=800.0 PL=0
MOVL C00369 V=800.0 PL=0
MOVL C00370 V=800.0 PL=0
MOVL C00371 V=800.0 PL=0
MOVL C00372 V=800.0 PL=0
MOVL C00373 V=800.0 PL=0
MOVL C00374 V=800.0 PL=0
MOVL C00375 V=800.0 PL=0
MOVL C00376 V=800.0 PL=0
MOVL C00377 V=800.0 PL=0
MOVL C00378 V=800.0 PL=0
MOVL C00379 V=800.0 PL=0
MOVL C00380 V=800.0 PL=0
MOVL C00381 V=800.0 PL=0
MOVL C00382 V=800.0 PL=0
MOVL C00383 V=800.0 PL=0
MOVL C00384 V=800.0 PL=0
MOVL C00385 V=800.0 PL=0
MOVL C00386 V=800.0 PL=0
MOVL C00387 V=800.0 PL=0
MOVL C00388 V=800.0 PL=0
MOVL C00389 V=800.0 PL=0
MOVL C00390 V=800.0 PL=0
MOVL C00391 V=800.0 PL=0
MOVL C00392 V=800.0 PL=0
MOVL C00393 V=800.0 PL=0
MOVL C00394 V=800.0 PL=0
MOVL C00395 V=800.0 PL=0
MOVL C00396 V=800.0 PL=0
MOVL C00397 V=800.0 PL=0
MOVL C00398 V=800.0 PL=0
MOVL C00399 V=800.0 PL=0
MOVL C00400 V=800.0 PL=0
MOVL C00401 V=800.0 PL=0
MOVL C00402 V=800.0 PL=0
MOVL C00403 V=800.0 PL=0
MOVL C00404 V=800.0 PL=0
MOVL C00405 V=800.0 PL=0
MOVL C00406 V=800.0 PL=0
MOVL C00407 V=800.0 PL=0
MOVL C00408 V=800.0 PL=0
MOVL C00409 V=800.0 PL=0
MOVL C00410 V=800.0 PL=0
MOVL C00411 V=800.0 PL=0
MOVL C00412 V=800.0 PL=0
MOVL C00413 V=800.0 PL=0
MOVL C00414 V=800.0 PL=0
MOVL C00415 V=800.0 PL=0
MOVL C00416 V=800.0 PL=0
MOVL C00417 V=800.0 PL=0
MOVL C00418 V=800.0 PL=0
MOVL C00419 V=800.0 PL=0
MOVL C00420 V=800.0 PL=0
MOVL C00421 V=800.0 PL=0
MOVL C00422 V=800.0 PL=0
MOVL C00423 V=800.0 PL=0
MOVL C00424 V=800.0 PL=0
MOVL C00425 V=800.0 PL=0
MOVL C00426 V=800.0 PL=0
MOVL C00427 V=800.0 PL=0
MOVL C00428 V=800.0 PL=0
MOVL C00429 V=800.0 PL=0
MOVL C00430 V=800.0 PL=0
MOVL C00431 V=800.0 PL=0
MOVL C00432 V=800.0 PL=0
MOVL C00433 V=800.0 PL=0
MOVL C00434 V=800.0 PL=0
MOVL C00435 V=800.0 PL=0
MOVL C00436 V=800.0 PL=0
MOVL C00437 V=800.0 PL=0
MOVL C00438 V=800.0 PL=0
MOVL C00439 V=800.0 PL=0
MOVL C00440 V=800.0 PL=0
MOVL C00441 V=800.0 PL=0
MOVL C00442 V=800.0 PL=0
MOVL C00443 V=800.0 PL=0
MOVL C00444 V=800.0 PL=0
MOVL C00445 V=800.0 PL=0
MOVL C00446 V=800.0 PL=0
MOVL C00447 V=800.0 PL=0
MOVL C00448 V=800.0 PL=0
MOVL C00449 V=800.0 PL=0
MOVL C00450 V=800.0 PL=0
MOVL C00451 V=800.0 PL=0
MOVL C00452 V=800.0 PL=0
MOVL C00453 V=800.0 PL=0
MOVL C00454 V=800.0 PL=0
MOVL C00455 V=800.0 PL=0
MOVL C00456 V=800.0 PL=0
MOVL C00457 V=800.0 PL=0
MOVL C00458 V=800.0 PL=0
MOVL C00459 V=800.0 PL=0
MOVL C00460 V=800.0 PL=0
MOVL C00461 V=800.0 PL=0
MOVL C00462 V=800.0 PL=0
MOVL C00463 V=800.0 PL=0
MOVL C00464 V=800.0 PL=0
MOVL C00465 V=800.0 PL=0
MOVL C00466 V=800.0 PL=0
MOVL C00467 V=800.0 PL=0
MOVL C00468 V=800.0 PL=0
MOVL C00469 V=800.0 PL=0
MOVL C00470 V=800.0 PL=0
MOVL C00471 V=800.0 PL=0
MOVL C00472 V=800.0 PL=0
MOVL C00473 V=800.0 PL=0
MOVL C00474 V=800.0 PL=0
MOVL C00475 V=800.0 PL=0
MOVL C00476 V=800.0 PL=0
MOVL C00477 V=800.0 PL=0
MOVL C00478 V=800.0 PL=0
MOVL C00479 V=800.0 PL=0
MOVL C00480 V=800.0 PL=0
MOVL C00481 V=800.0 PL=0
MOVL C00482 V=800.0 PL=0
MOVL C00483 V=800.0 PL=0
MOVL C00484 V=800.0 PL=0
MOVL C00485 V=800.0 PL=0
MOVL C00486 V=800.0 PL=0
MOVL C00487 V=800.0 PL=0
MOVL C00488 V=800.0 PL=0
MOVL C00489 V=800.0 PL=0
MOVL C00490 V=800.0 PL=0
MOVL C00491 V=800.0 PL=0
MOVL C00492 V=800.0 PL=0
MOVL C00493 V=800.0 PL=0
MOVL C00494 V=800.0 PL=0
MOVL C00495 V=800.0 PL=0
MOVL C00496 V=800.0 PL=0
MOVL C00497 V=800.0 PL=0
MOVL C00498 V=800.0 PL=0
MOVL C00499 V=800.0 PL=0
MOVL C00500 V=800.0 PL=0
MOVL C00501 V=800.0 PL=0
MOVL C00502 V=800.0 PL=0
MOVL C00503 V=800.0 PL=0
MOVL C00504 V=800.0 PL=0
MOVL C00505 V=800.0 PL=0
MOVL C00506 V=800.0 PL=0
MOVL C00507 V=800.0 PL=0
MOVL C00508 V=800.0 PL=0
MOVL C00509 V=800.0 PL=0
MOVL C00510 V=800.0 PL=0
MOVL C00511 V=800.0 PL=0
MOVL C00512 V=800.0 PL=0
MOVL C00513 V=800.0 PL=0
MOVL C00514 V=800.0 PL=0
MOVL C00515 V=800.0 PL=0
MOVL C00516 V=800.0 PL=0
MOVL C00517 V=800.0 PL=0
MOVL C00518 V=800.0 PL=0
MOVL C00519 V=800.0 PL=0
MOVL C00520 V=800.0 PL=0
MOVL C00521 V=800.0 PL=0
MOVL C00522 V=800.0 PL=0
MOVL C00523 V=800.0 PL=0
MOVL C00524 V=800.0 PL=0
MOVL C00525 V=800.0 PL=0
MOVL C00526 V=800.0 PL=0
MOVL C00527 V=800.0 PL=0
MOVL C00528 V=800.0 PL=0
MOVL C00529 V=800.0 PL=0
MOVL C00530 V=800.0 PL=0
MOVL C00531 V=800.0 PL=0
MOVL C00532 V=800.0 PL=0
MOVL C00533 V=800.0 PL=0
MOVL C00534 V=800.0 PL=0
MOVL C00535 V=800.0 PL=0
MOVL C00536 V=800.0 PL=0
MOVL C00537 V=800.0 PL=0
MOVL C00538 V=800.0 PL=0
MOVL C00539 V=800.0 PL=0
MOVL C00540 V=800.0 PL=0
MOVL C00541 V=800.0 PL=0
MOVL C00542 V=800.0 PL=0
MOVL C00543 V=800.0 PL=0
MOVL C00544 V=800.0 PL=0
MOVL C00545 V=800.0 PL=0
MOVL C00546 V=800.0 PL=0
MOVL C00547 V=800.0 PL=0
MOVL C00548 V=800.0 PL=0
MOVL C00549 V=800.0 PL=0
MOVL C00550 V=800.0 PL=0
MOVL C00551 V=800.0 PL=0
MOVL C00552 V=800.0 PL=0
MOVL C00553 V=800.0 PL=0
MOVL C00554 V=800.0 PL=0
MOVL C00555 V=800.0 PL=0
MOVL C00556 V=800.0 PL=0
MOVL C00557 V=800.0 PL=0
MOVL C00558 V=800.0 PL=0
MOVL C00559 V=800.0 PL=0
MOVL C00560 V=800.0 PL=0
MOVL C00561 V=800.0 PL=0
MOVL C00562 V=800.0 PL=0
MOVL C00563 V=800.0 PL=0
MOVL C00564 V=800.0 PL=0
MOVL C00565 V=800.0 PL=0
MOVL C00566 V=800.0 PL=0
MOVL C00567 V=800.0 PL=0
MOVL C00568 V=800.0 PL=0
MOVL C00569 V=800.0 PL=0
MOVL C00570 V=800.0 PL=0
MOVL C00571 V=800.0 PL=0
MOVL C00572 V=800.0 PL=0
MOVL C00573 V=800.0 PL=0
MOVL C00574 V=800.0 PL=0
MOVL C00575 V=800.0 PL=0
MOVL C00576 V=800.0 PL=0
MOVL C00577 V=800.0 PL=0
MOVL C00578 V=800.0 PL=0
MOVL C00579 V=800.0 PL=0
MOVL C00580 V=800.0 PL=0
MOVL C00581 V=800.0 PL=0
MOVL C00582 V=800.0 PL=0
MOVL C00583 V=800.0 PL=0
MOVL C00584 V=800.0 PL=0
MOVL C00585 V=800.0 PL=0
MOVL C00586 V=800.0 PL=0
MOVL C00587 V=800.0 PL=0
MOVL C00588 V=800.0 PL=0
MOVL C00589 V=800.0 PL=0
MOVL C00590 V=800.0 PL=0
MOVL C00591 V=800.0 PL=0
MOVL C00592 V=800.0 PL=0
MOVL C00593 V=800.0 PL=0
MOVL C00594 V=800.0 PL=0
MOVL C00595 V=800.0 PL=0
MOVL C00596 V=800.0 PL=0
MOVL C00597 V=800.0 PL=0
MOVL C00598 V=800.0 PL=0
MOVL C00599 V=800.0 PL=0
MOVL C00600 V=800.0 PL=0
MOVL C00601 V=800.0 PL=0
MOVL C00602 V=800.0 PL=0
MOVL C00603 V=800.0 PL=0
MOVL C00604 V=800.0 PL=0
MOVL C00605 V=800.0 PL=0
MOVL C00606 V=800.0 PL=0
MOVL C00607 V=800.0 PL=0
MOVL C00608 V=800.0 PL=0
MOVL C00609 V=800.0 PL=0
MOVL C00610 V=800.0 PL=0
MOVL C00611 V=800.0 PL=0
MOVL C00612 V=800.0 PL=0
MOVL C00613 V=800.0 PL=0
MOVL C00614 V=800.0 PL=0
MOVL C00615 V=800.0 PL=0
MOVL C00616 V=800.0 PL=0
MOVL C00617 V=800.0 PL=0
MOVL C00618 V=800.0 PL=0
MOVL C00619 V=800.0 PL=0
MOVL C00620 V=800.0 PL=0
MOVL C00621 V=800.0 PL=0
MOVL C00622 V=800.0 PL=0
MOVL C00623 V=800.0 PL=0
MOVL C00624 V=800.0 PL=0
MOVL C00625 V=800.0 PL=0
MOVL C00626 V=800.0 PL=0
MOVL C00627 V=800.0 PL=0
MOVL C00628 V=800.0 PL=0
MOVL C00629 V=800.0 PL=0
MOVL C00630 V=800.0 PL=0
MOVL C00631 V=800.0 PL=0
MOVL C00632 V=800.0 PL=0
MOVL C00633 V=800.0 PL=0
MOVL C00634 V=800.0 PL=0
MOVL C00635 V=800.0 PL=0
MOVL C00636 V=800.0 PL=0
MOVL C00637 V=800.0 PL=0
MOVL C00638 V=800.0 PL=0
MOVL C00639 V=800.0 PL=0
MOVL C00640 V=800.0 PL=0
MOVL C00641 V=800.0 PL=0
MOVL C00642 V=800.0 PL=0
MOVL C00643 V=800.0 PL=0
MOVL C00644 V=800.0 PL=0
MOVL C00645 V=800.0 PL=0
MOVL C00646 V=800.0 PL=0
MOVL C00647 V=800.0 PL=0
MOVL C00648 V=800.0 PL=0
MOVL C00649 V=800.0 PL=0
MOVL C00650 V=800.0 PL=0
MOVL C00651 V=800.0 PL=0
MOVL C00652 V=800.0 PL=0
MOVL C00653 V=800.0 PL=0
MOVL C00654 V=800.0 PL=0
MOVL C00655 V=800.0 PL=0
MOVL C00656 V=800.0 PL=0
MOVL C00657 V=800.0 PL=0
MOVL C00658 V=800.0 PL=0
MOVL C00659 V=800.0 PL=0
MOVL C00660 V=800.0 PL=0
MOVL C00661 V=800.0 PL=0
MOVL C00662 V=800.0 PL=0
MOVL C00663 V=800.0 PL=0
MOVL C00664 V=800.0 PL=0
MOVL C00665 V=800.0 PL=0
MOVL C00666 V=800.0 PL=0
MOVL C00667 V=800.0 PL=0
MOVL C00668 V=800.0 PL=0
MOVL C00669 V=800.0 PL=0
MOVL C00670 V=800.0 PL=0
MOVL C00671 V=800.0 PL=0
MOVL C00672 V=800.0 PL=0
MOVL C00673 V=800.0 PL=0
MOVL C00674 V=800.0 PL=0
MOVL C00675 V=800.0 PL=0
MOVL C00676 V=800.0 PL=0
MOVL C00677 V=800.0 PL=0
MOVL C00678 V=800.0 PL=0
MOVL C00679 V=800.0 PL=0
MOVL C00680 V=800.0 PL=0
MOVL C00681 V=800.0 PL=0
MOVL C00682 V=800.0 PL=0
MOVL C00683 V=800.0 PL=0
MOVL C00684 V=800.0 PL=0
MOVL C00685 V=800.0 PL=0
MOVL C00686 V=800.0 PL=0
MOVL C00687 V=800.0 PL=0
MOVL C00688 V=800.0 PL=0
MOVL C00689 V=800.0 PL=0
MOVL C00690 V=800.0 PL=0
MOVL C00691 V=800.0 PL=0
MOVL C00692 V=800.0 PL=0
MOVL C00693 V=800.0 PL=0
MOVL C00694 V=800.0 PL=0
MOVL C00695 V=800.0 PL=0
MOVL C00696 V=800.0 PL=0
MOVL C00697 V=800.0 PL=0
MOVL C00698 V=800.0 PL=0
MOVL C00699 V=800.0 PL=0
MOVL C00700 V=800.0 PL=0
MOVL C00701 V=800.0 PL=0
MOVL C00702 V=800.0 PL=0
MOVL C00703 V=800.0 PL=0
MOVL C00704 V=800.0 PL=0
MOVL C00705 V=800.0 PL=0
MOVL C00706 V=800.0 PL=0
MOVL C00707 V=800.0 PL=0
MOVL C00708 V=800.0 PL=0
MOVL C00709 V=800.0 PL=0
MOVL C00710 V=800.0 PL=0
MOVL C00711 V=800.0 PL=0
MOVL C00712 V=800.0 PL=0
MOVL C00713 V=800.0 PL=0
MOVL C00714 V=800.0 PL=0
MOVL C00715 V=800.0 PL=0
MOVL C00716 V=800.0 PL=0
MOVL C00717 V=800.0 PL=0
MOVL C00718 V=800.0 PL=0
MOVL C00719 V=800.0 PL=0
MOVL C00720 V=800.0 PL=0
MOVL C00721 V=800.0 PL=0
MOVL C00722 V=800.0 PL=0
MOVL C00723 V=800.0 PL=0
MOVL C00724 V=800.0 PL=0
MOVL C00725 V=800.0 PL=0
MOVL C00726 V=800.0 PL=0
MOVL C00727 V=800.0 PL=0
MOVL C00728 V=800.0 PL=0
MOVL C00729 V=800.0 PL=0
MOVL C00730 V=800.0 PL=0
MOVL C00731 V=800.0 PL=0
MOVL C00732 V=800.0 PL=0
MOVL C00733 V=800.0 PL=0
MOVL C00734 V=800.0 PL=0
MOVL C00735 V=800.0 PL=0
MOVL C00736 V=800.0 PL=0
MOVL C00737 V=800.0 PL=0
MOVL C00738 V=800.0 PL=0
MOVL C00739 V=800.0 PL=0
MOVL C00740 V=800.0 PL=0
MOVL C00741 V=800.0 PL=0
MOVL C00742 V=800.0 PL=0
MOVL C00743 V=800.0 PL=0
MOVL C00744 V=800.0 PL=0
MOVL C00745 V=800.0 PL=0
MOVL C00746 V=800.0 PL=0
MOVL C00747 V=800.0 PL=0
MOVL C00748 V=800.0 PL=0
MOVL C00749 V=800.0 PL=0
MOVL C00750 V=800.0 PL=0
MOVL C00751 V=800.0 PL=0
MOVL C00752 V=800.0 PL=0
MOVL C00753 V=800.0 PL=0
MOVL C00754 V=800.0 PL=0
MOVL C00755 V=800.0 PL=0
MOVL C00756 V=800.0 PL=0
MOVL C00757 V=800.0 PL=0
MOVL C00758 V=800.0 PL=0
MOVL C00759 V=800.0 PL=0
MOVL C00760 V=800.0 PL=0
MOVL C00761 V=800.0 PL=0
MOVL C00762 V=800.0 PL=0
MOVL C00763 V=800.0 PL=0
MOVL C00764 V=800.0 PL=0
MOVL C00765 V=800.0 PL=0
MOVL C00766 V=800.0 PL=0
MOVL C00767 V=800.0 PL=0
MOVL C00768 V=800.0 PL=0
MOVL C00769 V=800.0 PL=0
MOVL C00770 V=800.0 PL=0
MOVL C00771 V=800.0 PL=0
MOVL C00772 V=800.0 PL=0
MOVL C00773 V=800.0 PL=0
MOVL C00774 V=800.0 PL=0
MOVL C00775 V=800.0 PL=0
MOVL C00776 V=800.0 PL=0
MOVL C00777 V=800.0 PL=0
MOVL C00778 V=800.0 PL=0
MOVL C00779 V=800.0 PL=0
MOVL C00780 V=800.0 PL=0
MOVL C00781 V=800.0 PL=0
MOVL C00782 V=800.0 PL=0
MOVL C00783 V=800.0 PL=0
MOVL C00784 V=800.0 PL=0
MOVL C00785 V=800.0 PL=0
MOVL C00786 V=800.0 PL=0
MOVL C00787 V=800.0 PL=0
MOVL C00788 V=800.0 PL=0
MOVL C00789 V=800.0 PL=0
MOVL C00790 V=800.0 PL=0
MOVL C00791 V=800.0 PL=0
MOVL C00792 V=800.0 PL=0
MOVL C00793 V=800.0 PL=0
MOVL C00794 V=800.0 PL=0
MOVL C00795 V=800.0 PL=0
MOVL C00796 V=800.0 PL=0
MOVL C00797 V=800.0 PL=0
MOVL C00798 V=800.0 PL=0
MOVL C00799 V=800.0 PL=0
MOVL C00800 V=800.0 PL=0
MOVL C00801 V=800.0 PL=0
MOVL C00802 V=800.0 PL=0
MOVL C00803 V=800.0 PL=0
MOVL C00804 V=800.0 PL=0
MOVL C00805 V=800.0 PL=0
MOVL C00806 V=800.0 PL=0
MOVL C00807 V=800.0 PL=0
MOVL C00808 V=800.0 PL=0
MOVL C00809 V=800.0 PL=0
MOVL C00810 V=800.0 PL=0
MOVL C00811 V=800.0 PL=0
MOVL C00812 V=800.0 PL=0
MOVL C00813 V=800.0 PL=0
MOVL C00814 V=800.0 PL=0
MOVL C00815 V=800.0 PL=0
MOVL C00816 V=800.0 PL=0
MOVL C00817 V=800.0 PL=0
MOVL C00818 V=800.0 PL=0
MOVL C00819 V=800.0 PL=0
MOVL C00820 V=800.0 PL=0
MOVL C00821 V=800.0 PL=0
MOVL C00822 V=800.0 PL=0
MOVL C00823 V=800.0 PL=0
MOVL C00824 V=800.0 PL=0
MOVL C00825 V=800.0 PL=0
MOVL C00826 V=800.0 PL=0
MOVL C00827 V=800.0 PL=0
MOVL C00828 V=800.0 PL=0
MOVL C00829 V=800.0 PL=0
MOVL C00830 V=800.0 PL=0
MOVL C00831 V=800.0 PL=0
MOVL C00832 V=800.0 PL=0
MOVL C00833 V=800.0 PL=0
MOVL C00834 V=800.0 PL=0
MOVL C00835 V=800.0 PL=0
MOVL C00836 V=800.0 PL=0
MOVL C00837 V=800.0 PL=0
MOVL C00838 V=800.0 PL=0
MOVL C00839 V=800.0 PL=0
MOVL C00840 V=800.0 PL=0
MOVL C00841 V=800.0 PL=0
MOVL C00842 V=800.0 PL=0
MOVL C00843 V=800.0 PL=0
MOVL C00844 V=800.0 PL=0
MOVL C00845 V=800.0 PL=0
MOVL C00846 V=800.0 PL=0
MOVL C00847 V=800.0 PL=0
MOVL C00848 V=800.0 PL=0
MOVL C00849 V=800.0 PL=0
MOVL C00850 V=800.0 PL=0
MOVL C00851 V=800.0 PL=0
MOVL C00852 V=800.0 PL=0
MOVL C00853 V=800.0 PL=0
MOVL C00854 V=800.0 PL=0
MOVL C00855 V=800.0 PL=0
MOVL C00856 V=800.0 PL=0
MOVL C00857 V=800.0 PL=0
MOVL C00858 V=800.0 PL=0
MOVL C00859 V=800.0 PL=0
MOVL C00860 V=800.0 PL=0
MOVL C00861 V=800.0 PL=0
MOVL C00862 V=800.0 PL=0
MOVL C00863 V=800.0 PL=0
MOVL C00864 V=800.0 PL=0
MOVL C00865 V=800.0 PL=0
MOVL C00866 V=800.0 PL=0
MOVL C00867 V=800.0 PL=0
MOVL C00868 V=800.0 PL=0
MOVL C00869 V=800.0 PL=0
MOVL C00870 V=800.0 PL=0
MOVL C00871 V=800.0 PL=0
MOVL C00872 V=800.0 PL=0
MOVL C00873 V=800.0 PL=0
MOVL C00874 V=800.0 PL=0
MOVL C00875 V=800.0 PL=0
MOVL C00876 V=800.0 PL=0
MOVL C00877 V=800.0 PL=0
MOVL C00878 V=800.0 PL=0
MOVL C00879 V=800.0 PL=0
MOVL C00880 V=800.0 PL=0
MOVL C00881 V=800.0 PL=0
MOVL C00882 V=800.0 PL=0
MOVL C00883 V=800.0 PL=0
MOVL C00884 V=800.0 PL=0
MOVL C00885 V=800.0 PL=0
MOVL C00886 V=800.0 PL=0
MOVL C00887 V=800.0 PL=0
MOVL C00888 V=800.0 PL=0
MOVL C00889 V=800.0 PL=0
MOVL C00890 V=800.0 PL=0
MOVL C00891 V=800.0 PL=0
MOVL C00892 V=800.0 PL=0
MOVL C00893 V=800.0 PL=0
MOVL C00894 V=800.0 PL=0
MOVL C00895 V=800.0 PL=0
MOVL C00896 V=800.0 PL=0
MOVL C00897 V=800.0 PL=0
MOVL C00898 V=800.0 PL=0
MOVL C00899 V=800.0 PL=0
MOVL C00900 V=800.0 PL=0
MOVL C00901 V=800.0 PL=0
MOVL C00902 V=800.0 PL=0
MOVL C00903 V=800.0 PL=0
MOVL C00904 V=800.0 PL=0
MOVL C00905 V=800.0 PL=0
MOVL C00906 V=800.0 PL=0
MOVL C00907 V=800.0 PL=0
MOVL C00908 V=800.0 PL=0
MOVL C00909 V=800.0 PL=0
MOVL C00910 V=800.0 PL=0
MOVL C00911 V=800.0 PL=0
MOVL C00912 V=800.0 PL=0
MOVL C00913 V=800.0 PL=0
MOVL C00914 V=800.0 PL=0
MOVL C00915 V=800.0 PL=0
MOVL C00916 V=800.0 PL=0
MOVL C00917 V=800.0 PL=0
MOVL C00918 V=800.0 PL=0
MOVL C00919 V=800.0 PL=0
MOVL C00920 V=800.0 PL=0
MOVL C00921 V=800.0 PL=0
MOVL C00922 V=800.0 PL=0
MOVL C00923 V=800.0 PL=0
MOVL C00924 V=800.0 PL=0
MOVL C00925 V=800.0 PL=0
MOVL C00926 V=800.0 PL=0
MOVL C00927 V=800.0 PL=0
MOVL C00928 V=800.0 PL=0
MOVL C00929 V=800.0 PL=0
MOVL C00930 V=800.0 PL=0
MOVL C00931 V=800.0 PL=0
MOVL C00932 V=800.0 PL=0
MOVL C00933 V=800.0 PL=0
MOVL C00934 V=800.0 PL=0
MOVL C00935 V=800.0 PL=0
MOVL C00936 V=800.0 PL=0
MOVL C00937 V=800.0 PL=0
MOVL C00938 V=800.0 PL=0
MOVL C00939 V=800.0 PL=0
MOVL C00940 V=800.0 PL=0
MOVL C00941 V=800.0 PL=0
MOVL C00942 V=800.0 PL=0
MOVL C00943 V=800.0 PL=0
MOVL C00944 V=800.0 PL=0
MOVL C00945 V=800.0 PL=0
MOVL C00946 V=800.0 PL=0
MOVL C00947 V=800.0 PL=0
MOVL C00948 V=800.0 PL=0
MOVL C00949 V=800.0 PL=0
MOVL C00950 V=800.0 PL=0
MOVL C00951 V=800.0 PL=0
MOVL C00952 V=800.0 PL=0
MOVL C00953 V=800.0 PL=0
MOVL C00954 V=800.0 PL=0
MOVL C00955 V=800.0 PL=0
MOVL C00956 V=800.0 PL=0
MOVL C00957 V=800.0 PL=0
MOVL C00958 V=800.0 PL=0
MOVL C00959 V=800.0 PL=0
MOVL C00960 V=800.0 PL=0
MOVL C00961 V=800.0 PL=0
MOVL C00962 V=800.0 PL=0
MOVL C00963 V=800.0 PL=0
MOVL C00964 V=800.0 PL=0
MOVL C00965 V=800.0 PL=0
MOVL C00966 V=800.0 PL=0
MOVL C00967 V=800.0 PL=0
MOVL C00968 V=800.0 PL=0
MOVL C00969 V=800.0 PL=0
MOVL C00970 V=800.0 PL=0
MOVL C00971 V=800.0 PL=0
MOVL C00972 V=800.0 PL=0
MOVL C00973 V=800.0 PL=0
MOVL C00974 V=800.0 PL=0
MOVL C00975 V=800.0 PL=0
MOVL C00976 V=800.0 PL=0
MOVL C00977 V=800.0 PL=0
MOVL C00978 V=800.0 PL=0
MOVL C00979 V=800.0 PL=0
MOVL C00980 V=800.0 PL=0
MOVL C00981 V=800.0 PL=0
MOVL C00982 V=800.0 PL=0
MOVL C00983 V=800.0 PL=0
MOVL C00984 V=800.0 PL=0
MOVL C00985 V=800.0 PL=0
MOVL C00986 V=800.0 PL=0
MOVL C00987 V=800.0 PL=0
MOVL C00988 V=800.0 PL=0
MOVL C00989 V=800.0 PL=0
MOVL C00990 V=800.0 PL=0
MOVL C00991 V=800.0 PL=0
MOVL C00992 V=800.0 PL=0
MOVL C00993 V=800.0 PL=0
MOVL C00994 V=800.0 PL=0
MOVL C00995 V=800.0 PL=0
MOVL C00996 V=800.0 PL=0
MOVL C00997 V=800.0 PL=0
MOVL C00998 V=800.0 PL=0
MOVL C00999 V=800.0 PL=0
MOVL C01000 V=800.0 PL=0
MOVL C01001 V=800.0 PL=0
MOVL C01002 V=800.0 PL=0
MOVL C01003 V=800.0 PL=0
MOVL C01004 V=800.0 PL=0
MOVL C01005 V=800.0 PL=0
MOVL C01006 V=800.0 PL=0
MOVL C01007 V=800.0 PL=0
MOVL C01008 V=800.0 PL=0
MOVL C01009 V=800.0 PL=0
MOVL C01010 V=800.0 PL=0
MOVL C01011 V=800.0 PL=0
MOVL C01012 V=800.0 PL=0
MOVL C01013 V=800.0 PL=0
MOVL C01014 V=800.0 PL=0
MOVL C01015 V=800.0 PL=0
MOVL C01016 V=800.0 PL=0
MOVL C01017 V=800.0 PL=0
MOVL C01018 V=800.0 PL=0
MOVL C01019 V=800.0 PL=0
MOVL C01020 V=800.0 PL=0
MOVL C01021 V=800.0 PL=0
MOVL C01022 V=800.0 PL=0
MOVL C01023 V=800.0 PL=0
MOVL C01024 V=800.0 PL=0
MOVL C01025 V=800.0 PL=0
MOVL C01026 V=800.0 PL=0
MOVL C01027 V=800.0 PL=0
MOVL C01028 V=800.0 PL=0
MOVL C01029 V=800.0 PL=0
MOVL C01030 V=800.0 PL=0
MOVL C01031 V=800.0 PL=0
MOVL C01032 V=800.0 PL=0
MOVL C01033 V=800.0 PL=0
MOVL C01034 V=800.0 PL=0
MOVL C01035 V=800.0 PL=0
MOVL C01036 V=800.0 PL=0
MOVL C01037 V=800.0 PL=0
MOVL C01038 V=800.0 PL=0
MOVL C01039 V=800.0 PL=0
MOVL C01040 V=800.0 PL=0
MOVL C01041 V=800.0 PL=0
MOVL C01042 V=800.0 PL=0
MOVL C01043 V=800.0 PL=0
MOVL C01044 V=800.0 PL=0
MOVL C01045 V=800.0 PL=0
MOVL C01046 V=800.0 PL=0
MOVL C01047 V=800.0 PL=0
MOVL C01048 V=800.0 PL=0
MOVL C01049 V=800.0 PL=0
MOVL C01050 V=800.0 PL=0
MOVL C01051 V=800.0 PL=0
MOVL C01052 V=800.0 PL=0
MOVL C01053 V=800.0 PL=0
MOVL C01054 V=800.0 PL=0
MOVL C01055 V=800.0 PL=0
MOVL C01056 V=800.0 PL=0
MOVL C01057 V=800.0 PL=0
MOVL C01058 V=800.0 PL=0
MOVL C01059 V=800.0 PL=0
MOVL C01060 V=800.0 PL=0
MOVL C01061 V=800.0 PL=0
MOVL C01062 V=800.0 PL=0
MOVL C01063 V=800.0 PL=0
MOVL C01064 V=800.0 PL=0
MOVL C01065 V=800.0 PL=0
MOVL C01066 V=800.0 PL=0
MOVL C01067 V=800.0 PL=0
MOVL C01068 V=800.0 PL=0
MOVL C01069 V=800.0 PL=0
MOVL C01070 V=800.0 PL=0
MOVL C01071 V=800.0 PL=0
MOVL C01072 V=800.0 PL=0
MOVL C01073 V=800.0 PL=0
MOVL C01074 V=800.0 PL=0
MOVL C01075 V=800.0 PL=0
MOVL C01076 V=800.0 PL=0
MOVL C01077 V=800.0 PL=0
MOVL C01078 V=800.0 PL=0
MOVL C01079 V=800.0 PL=0
MOVL C01080 V=800.0 PL=0
MOVL C01081 V=800.0 PL=0
MOVL C01082 V=800.0 PL=0
MOVL C01083 V=800.0 PL=0
MOVL C01084 V=800.0 PL=0
MOVL C01085 V=800.0 PL=0
MOVL C01086 V=800.0 PL=0
MOVL C01087 V=800.0 PL=0
MOVL C01088 V=800.0 PL=0
MOVL C01089 V=800.0 PL=0
MOVL C01090 V=800.0 PL=0
MOVL C01091 V=800.0 PL=0
MOVL C01092 V=800.0 PL=0
MOVL C01093 V=800.0 PL=0
MOVL C01094 V=800.0 PL=0
MOVL C01095 V=800.0 PL=0
MOVL C01096 V=800.0 PL=0
MOVL C01097 V=800.0 PL=0
MOVL C01098 V=800.0 PL=0
MOVL C01099 V=800.0 PL=0
MOVL C01100 V=800.0 PL=0
MOVL C01101 V=800.0 PL=0
MOVL C01102 V=800.0 PL=0
MOVL C01103 V=800.0 PL=0
MOVL C01104 V=800.0 PL=0
MOVL C01105 V=800.0 PL=0
MOVL C01106 V=800.0 PL=0
MOVL C01107 V=800.0 PL=0
MOVL C01108 V=800.0 PL=0
MOVL C01109 V=800.0 PL=0
MOVL C01110 V=800.0 PL=0
MOVL C01111 V=800.0 PL=0
MOVL C01112 V=800.0 PL=0
MOVL C01113 V=800.0 PL=0
MOVL C01114 V=800.0 PL=0
MOVL C01115 V=800.0 PL=0
MOVL C01116 V=800.0 PL=0
MOVL C01117 V=800.0 PL=0
MOVL C01118 V=800.0 PL=0
MOVL C01119 V=800.0 PL=0
MOVL C01120 V=800.0 PL=0
MOVL C01121 V=800.0 PL=0
MOVL C01122 V=800.0 PL=0
MOVL C01123 V=800.0 PL=0
MOVL C01124 V=800.0 PL=0
MOVL C01125 V=800.0 PL=0
MOVL C01126 V=800.0 PL=0
MOVL C01127 V=800.0 PL=0
MOVL C01128 V=800.0 PL=0
MOVL C01129 V=800.0 PL=0
MOVL C01130 V=800.0 PL=0
MOVL C01131 V=800.0 PL=0
MOVL C01132 V=800.0 PL=0
MOVL C01133 V=800.0 PL=0
MOVL C01134 V=800.0 PL=0
MOVL C01135 V=800.0 PL=0
MOVL C01136 V=800.0 PL=0
MOVL C01137 V=800.0 PL=0
MOVL C01138 V=800.0 PL=0
MOVL C01139 V=800.0 PL=0
MOVL C01140 V=800.0 PL=0
MOVL C01141 V=800.0 PL=0
MOVL C01142 V=800.0 PL=0
MOVL C01143 V=800.0 PL=0
MOVL C01144 V=800.0 PL=0
MOVL C01145 V=800.0 PL=0
MOVL C01146 V=800.0 PL=0
MOVL C01147 V=800.0 PL=0
MOVL C01148 V=800.0 PL=0
MOVL C01149 V=800.0 PL=0
MOVL C01150 V=800.0 PL=0
MOVL C01151 V=800.0 PL=0
MOVL C01152 V=800.0 PL=0
MOVL C01153 V=800.0 PL=0
MOVL C01154 V=800.0 PL=0
MOVL C01155 V=800.0 PL=0
MOVL C01156 V=800.0 PL=0
MOVL C01157 V=800.0 PL=0
MOVL C01158 V=800.0 PL=0
MOVL C01159 V=800.0 PL=0
MOVL C01160 V=800.0 PL=0
MOVL C01161 V=800.0 PL=0
MOVL C01162 V=800.0 PL=0
MOVL C01163 V=800.0 PL=0
MOVL C01164 V=800.0 PL=0
MOVL C01165 V=800.0 PL=0
MOVL C01166 V=800.0 PL=0
MOVL C01167 V=800.0 PL=0
MOVL C01168 V=800.0 PL=0
MOVL C01169 V=800.0 PL=0
MOVL C01170 V=800.0 PL=0
MOVL C01171 V=800.0 PL=0
MOVL C01172 V=800.0 PL=0
MOVL C01173 V=800.0 PL=0
MOVL C01174 V=800.0 PL=0
MOVL C01175 V=800.0 PL=0
MOVL C01176 V=800.0 PL=0
MOVL C01177 V=800.0 PL=0
MOVL C01178 V=800.0 PL=0
MOVL C01179 V=800.0 PL=0
MOVL C01180 V=800.0 PL=0
MOVL C01181 V=800.0 PL=0
MOVL C01182 V=800.0 PL=0
MOVL C01183 V=800.0 PL=0
MOVL C01184 V=800.0 PL=0
MOVL C01185 V=800.0 PL=0
MOVL C01186 V=800.0 PL=0
MOVL C01187 V=800.0 PL=0
MOVL C01188 V=800.0 PL=0
MOVL C01189 V=800.0 PL=0
MOVL C01190 V=800.0 PL=0
MOVL C01191 V=800.0 PL=0
MOVL C01192 V=800.0 PL=0
MOVL C01193 V=800.0 PL=0
MOVL C01194 V=800.0 PL=0
MOVL C01195 V=800.0 PL=0
MOVL C01196 V=800.0 PL=0
MOVL C01197 V=800.0 PL=0
MOVL C01198 V=800.0 PL=0
MOVL C01199 V=800.0 PL=0
MOVL C01200 V=800.0 PL=0
MOVL C01201 V=800.0 PL=0
MOVL C01202 V=800.0 PL=0
MOVL C01203 V=800.0 PL=0
MOVL C01204 V=800.0 PL=0
MOVL C01205 V=800.0 PL=0
MOVL C01206 V=800.0 PL=0
MOVL C01207 V=800.0 PL=0
MOVL C01208 V=800.0 PL=0
MOVL C01209 V=800.0 PL=0
MOVL C01210 V=800.0 PL=0
MOVL C01211 V=800.0 PL=0
MOVL C01212 V=800.0 PL=0
MOVL C01213 V=800.0 PL=0
MOVL C01214 V=800.0 PL=0
MOVL C01215 V=800.0 PL=0
MOVL C01216 V=800.0 PL=0
MOVL C01217 V=800.0 PL=0
MOVL C01218 V=800.0 PL=0
MOVL C01219 V=800.0 PL=0
MOVL C01220 V=800.0 PL=0
MOVL C01221 V=800.0 PL=0
MOVL C01222 V=800.0 PL=0
MOVL C01223 V=800.0 PL=0
MOVL C01224 V=800.0 PL=0
MOVL C01225 V=800.0 PL=0
MOVL C01226 V=800.0 PL=0
MOVL C01227 V=800.0 PL=0
MOVL C01228 V=800.0 PL=0
MOVL C01229 V=800.0 PL=0
MOVL C01230 V=800.0 PL=0
MOVL C01231 V=800.0 PL=0
MOVL C01232 V=800.0 PL=0
MOVL C01233 V=800.0 PL=0
MOVL C01234 V=800.0 PL=0
MOVL C01235 V=800.0 PL=0
MOVL C01236 V=800.0 PL=0
MOVL C01237 V=800.0 PL=0
MOVL C01238 V=800.0 PL=0
MOVL C01239 V=800.0 PL=0
MOVL C01240 V=800.0 PL=0
MOVL C01241 V=800.0 PL=0
MOVL C01242 V=800.0 PL=0
MOVL C01243 V=800.0 PL=0
MOVL C01244 V=800.0 PL=0
MOVL C01245 V=800.0 PL=0
MOVL C01246 V=800.0 PL=0
MOVL C01247 V=800.0 PL=0
MOVL C01248 V=800.0 PL=0
MOVL C01249 V=800.0 PL=0
MOVL C01250 V=800.0 PL=0
MOVL C01251 V=800.0 PL=0
MOVL C01252 V=800.0 PL=0
MOVL C01253 V=800.0 PL=0
MOVL C01254 V=800.0 PL=0
MOVL C01255 V=800.0 PL=0
MOVL C01256 V=800.0 PL=0
MOVL C01257 V=800.0 PL=0
MOVL C01258 V=800.0 PL=0
MOVL C01259 V=800.0 PL=0
MOVL C01260 V=800.0 PL=0
MOVL C01261 V=800.0 PL=0
MOVL C01262 V=800.0 PL=0
MOVL C01263 V=800.0 PL=0
MOVL C01264 V=800.0 PL=0
MOVL C01265 V=800.0 PL=0
MOVL C01266 V=800.0 PL=0
MOVL C01267 V=800.0 PL=0
MOVL C01268 V=800.0 PL=0
MOVL C01269 V=800.0 PL=0
MOVL C01270 V=800.0 PL=0
MOVL C01271 V=800.0 PL=0
MOVL C01272 V=800.0 PL=0
MOVL C01273 V=800.0 PL=0
MOVL C01274 V=800.0 PL=0
MOVL C01275 V=800.0 PL=0
MOVL C01276 V=800.0 PL=0
MOVL C01277 V=800.0 PL=0
MOVL C01278 V=800.0 PL=0
MOVL C01279 V=800.0 PL=0
MOVL C01280 V=800.0 PL=0
MOVL C01281 V=800.0 PL=0
MOVL C01282 V=800.0 PL=0
MOVL C01283 V=800.0 PL=0
MOVL C01284 V=800.0 PL=0
MOVL C01285 V=800.0 PL=0
MOVL C01286 V=800.0 PL=0
MOVL C01287 V=800.0 PL=0
MOVL C01288 V=800.0 PL=0
MOVL C01289 V=800.0 PL=0
MOVL C01290 V=800.0 PL=0
MOVL C01291 V=800.0 PL=0
MOVL C01292 V=800.0 PL=0
MOVL C01293 V=800.0 PL=0
MOVL C01294 V=800.0 PL=0
MOVL C01295 V=800.0 PL=0
MOVL C01296 V=800.0 PL=0
MOVL C01297 V=800.0 PL=0
MOVL C01298 V=800.0 PL=0
MOVL C01299 V=800.0 PL=0
MOVL C01300 V=800.0 PL=0
MOVL C01301 V=800.0 PL=0
MOVL C01302 V=800.0 PL=0
MOVL C01303 V=800.0 PL=0
MOVL C01304 V=800.0 PL=0
MOVL C01305 V=800.0 PL=0
MOVL C01306 V=800.0 PL=0
MOVL C01307 V=800.0 PL=0
MOVL C01308 V=800.0 PL=0
MOVL C01309 V=800.0 PL=0
MOVL C01310 V=800.0 PL=0
MOVL C01311 V=800.0 PL=0
MOVL C01312 V=800.0 PL=0
MOVL C01313 V=800.0 PL=0
MOVL C01314 V=800.0 PL=0
MOVL C01315 V=800.0 PL=0
MOVL C01316 V=800.0 PL=0
MOVL C01317 V=800.0 PL=0
MOVL C01318 V=800.0 PL=0
MOVL C01319 V=800.0 PL=0
MOVL C01320 V=800.0 PL=0
MOVL C01321 V=800.0 PL=0
MOVL C01322 V=800.0 PL=0
MOVL C01323 V=800.0 PL=0
MOVL C01324 V=800.0 PL=0
MOVL C01325 V=800.0 PL=0
MOVL C01326 V=800.0 PL=0
MOVL C01327 V=800.0 PL=0
MOVL C01328 V=800.0 PL=0
MOVL C01329 V=800.0 PL=0
MOVL C01330 V=800.0 PL=0
MOVL C01331 V=800.0 PL=0
MOVL C01332 V=800.0 PL=0
MOVL C01333 V=800.0 PL=0
MOVL C01334 V=800.0 PL=0
MOVL C01335 V=800.0 PL=0
MOVL C01336 V=800.0 PL=0
MOVL C01337 V=800.0 PL=0
MOVL C01338 V=800.0 PL=0
MOVL C01339 V=800.0 PL=0
MOVL C01340 V=800.0 PL=0
MOVL C01341 V=800.0 PL=0
MOVL C01342 V=800.0 PL=0
MOVL C01343 V=800.0 PL=0
MOVL C01344 V=800.0 PL=0
MOVL C01345 V=800.0 PL=0
MOVL C01346 V=800.0 PL=0
MOVL C01347 V=800.0 PL=0
MOVL C01348 V=800.0 PL=0
MOVL C01349 V=800.0 PL=0
MOVL C01350 V=800.0 PL=0
MOVL C01351 V=800.0 PL=0
MOVL C01352 V=800.0 PL=0
MOVL C01353 V=800.0 PL=0
MOVL C01354 V=800.0 PL=0
MOVL C01355 V=800.0 PL=0
MOVL C01356 V=800.0 PL=0
MOVL C01357 V=800.0 PL=0
MOVL C01358 V=800.0 PL=0
MOVL C01359 V=800.0 PL=0
MOVL C01360 V=800.0 PL=0
MOVL C01361 V=800.0 PL=0
MOVL C01362 V=800.0 PL=0
MOVL C01363 V=800.0 PL=0
MOVL C01364 V=800.0 PL=0
MOVL C01365 V=800.0 PL=0
MOVL C01366 V=800.0 PL=0
MOVL C01367 V=800.0 PL=0
MOVL C01368 V=800.0 PL=0
MOVL C01369 V=800.0 PL=0
MOVL C01370 V=800.0 PL=0
MOVL C01371 V=800.0 PL=0
MOVL C01372 V=800.0 PL=0
MOVL C01373 V=800.0 PL=0
MOVL C01374 V=800.0 PL=0
MOVL C01375 V=800.0 PL=0
MOVL C01376 V=800.0 PL=0
MOVL C01377 V=800.0 PL=0
MOVL C01378 V=800.0 PL=0
MOVL C01379 V=800.0 PL=0
MOVL C01380 V=800.0 PL=0
MOVL C01381 V=800.0 PL=0
MOVL C01382 V=800.0 PL=0
MOVL C01383 V=800.0 PL=0
MOVL C01384 V=800.0 PL=0
MOVL C01385 V=800.0 PL=0
MOVL C01386 V=800.0 PL=0
MOVL C01387 V=800.0 PL=0
MOVL C01388 V=800.0 PL=0
MOVL C01389 V=800.0 PL=0
MOVL C01390 V=800.0 PL=0
MOVL C01391 V=800.0 PL=0
MOVL C01392 V=800.0 PL=0
MOVL C01393 V=800.0 PL=0
MOVL C01394 V=800.0 PL=0
MOVL C01395 V=800.0 PL=0
MOVL C01396 V=800.0 PL=0
MOVL C01397 V=800.0 PL=0
MOVL C01398 V=800.0 PL=0
MOVL C01399 V=800.0 PL=0
MOVL C01400 V=800.0 PL=0
MOVL C01401 V=800.0 PL=0
MOVL C01402 V=800.0 PL=0
MOVL C01403 V=800.0 PL=0
MOVL C01404 V=800.0 PL=0
MOVL C01405 V=800.0 PL=0
MOVL C01406 V=800.0 PL=0
MOVL C01407 V=800.0 PL=0
MOVL C01408 V=800.0 PL=0
MOVL C01409 V=800.0 PL=0
MOVL C01410 V=800.0 PL=0
MOVL C01411 V=800.0 PL=0
MOVL C01412 V=800.0 PL=0
MOVL C01413 V=800.0 PL=0
MOVL C01414 V=800.0 PL=0
MOVL C01415 V=800.0 PL=0
MOVL C01416 V=800.0 PL=0
MOVL C01417 V=800.0 PL=0
MOVL C01418 V=800.0 PL=0
MOVL C01419 V=800.0 PL=0
MOVL C01420 V=800.0 PL=0
MOVL C01421 V=800.0 PL=0
MOVL C01422 V=800.0 PL=0
MOVL C01423 V=800.0 PL=0
MOVL C01424 V=800.0 PL=0
MOVL C01425 V=800.0 PL=0
MOVL C01426 V=800.0 PL=0
MOVL C01427 V=800.0 PL=0
MOVL C01428 V=800.0 PL=0
MOVL C01429 V=800.0 PL=0
MOVL C01430 V=800.0 PL=0
MOVL C01431 V=800.0 PL=0
MOVL C01432 V=800.0 PL=0
MOVL C01433 V=800.0 PL=0
MOVL C01434 V=800.0 PL=0
MOVL C01435 V=800.0 PL=0
MOVL C01436 V=800.0 PL=0
MOVL C01437 V=800.0 PL=0
MOVL C01438 V=800.0 PL=0
MOVL C01439 V=800.0 PL=0
MOVL C01440 V=800.0 PL=0
MOVL C01441 V=800.0 PL=0
MOVL C01442 V=800.0 PL=0
MOVL C01443 V=800.0 PL=0
MOVL C01444 V=800.0 PL=0
MOVL C01445 V=800.0 PL=0
MOVL C01446 V=800.0 PL=0
MOVL C01447 V=800.0 PL=0
MOVL C01448 V=800.0 PL=0
MOVL C01449 V=800.0 PL=0
MOVL C01450 V=800.0 PL=0
MOVL C01451 V=800.0 PL=0
MOVL C01452 V=800.0 PL=0
MOVL C01453 V=800.0 PL=0
MOVL C01454 V=800.0 PL=0
MOVL C01455 V=800.0 PL=0
MOVL C01456 V=800.0 PL=0
MOVL C01457 V=800.0 PL=0
MOVL C01458 V=800.0 PL=0
MOVL C01459 V=800.0 PL=0
MOVL C01460 V=800.0 PL=0
MOVL C01461 V=800.0 PL=0
MOVL C01462 V=800.0 PL=0
MOVL C01463 V=800.0 PL=0
MOVL C01464 V=800.0 PL=0
MOVL C01465 V=800.0 PL=0
MOVL C01466 V=800.0 PL=0
MOVL C01467 V=800.0 PL=0
MOVL C01468 V=800.0 PL=0
MOVL C01469 V=800.0 PL=0
MOVL C01470 V=800.0 PL=0
MOVL C01471 V=800.0 PL=0
MOVL C01472 V=800.0 PL=0
MOVL C01473 V=800.0 PL=0
MOVL C01474 V=800.0 PL=0
MOVL C01475 V=800.0 PL=0
MOVL C01476 V=800.0 PL=0
MOVL C01477 V=800.0 PL=0
MOVL C01478 V=800.0 PL=0
MOVL C01479 V=800.0 PL=0
MOVL C01480 V=800.0 PL=0
MOVL C01481 V=800.0 PL=0
MOVL C01482 V=800.0 PL=0
MOVL C01483 V=800.0 PL=0
MOVL C01484 V=800.0 PL=0
MOVL C01485 V=800.0 PL=0
MOVL C01486 V=800.0 PL=0
MOVL C01487 V=800.0 PL=0
MOVL C01488 V=800.0 PL=0
MOVL C01489 V=800.0 PL=0
MOVL C01490 V=800.0 PL=0
MOVL C01491 V=800.0 PL=0
MOVL C01492 V=800.0 PL=0
MOVL C01493 V=800.0 PL=0
MOVL C01494 V=800.0 PL=0
MOVL C01495 V=800.0 PL=0
MOVL C01496 V=800.0 PL=0
MOVL C01497 V=800.0 PL=0
MOVL C01498 V=800.0 PL=0
MOVL C01499 V=800.0 PL=0
MOVL C01500 V=800.0 PL=0
MOVL C01501 V=800.0 PL=0
MOVL C01502 V=800.0 PL=0
MOVL C01503 V=800.0 PL=0
MOVL C01504 V=800.0 PL=0
MOVL C01505 V=800.0 PL=0
MOVL C01506 V=800.0 PL=0
MOVL C01507 V=800.0 PL=0
MOVL C01508 V=800.0 PL=0
MOVL C01509 V=800.0 PL=0
MOVL C01510 V=800.0 PL=0
MOVL C01511 V=800.0 PL=0
MOVL C01512 V=800.0 PL=0
MOVL C01513 V=800.0 PL=0
MOVL C01514 V=800.0 PL=0
MOVL C01515 V=800.0 PL=0
MOVL C01516 V=800.0 PL=0
MOVL C01517 V=800.0 PL=0
MOVL C01518 V=800.0 PL=0
MOVL C01519 V=800.0 PL=0
MOVL C01520 V=800.0 PL=0
MOVL C01521 V=800.0 PL=0
MOVL C01522 V=800.0 PL=0
MOVL C01523 V=800.0 PL=0
MOVL C01524 V=800.0 PL=0
MOVL C01525 V=800.0 PL=0
MOVL C01526 V=800.0 PL=0
MOVL C01527 V=800.0 PL=0
MOVL C01528 V=800.0 PL=0
MOVL C01529 V=800.0 PL=0
MOVL C01530 V=800.0 PL=0
MOVL C01531 V=800.0 PL=0
MOVL C01532 V=800.0 PL=0
MOVL C01533 V=800.0 PL=0
MOVL C01534 V=800.0 PL=0
MOVL C01535 V=800.0 PL=0
MOVL C01536 V=800.0 PL=0
MOVL C01537 V=800.0 PL=0
MOVL C01538 V=800.0 PL=0
MOVL C01539 V=800.0 PL=0
MOVL C01540 V=800.0 PL=0
MOVL C01541 V=800.0 PL=0
MOVL C01542 V=800.0 PL=0
MOVL C01543 V=800.0 PL=0
MOVL C01544 V=800.0 PL=0
MOVL C01545 V=800.0 PL=0
MOVL C01546 V=800.0 PL=0
MOVL C01547 V=800.0 PL=0
MOVL C01548 V=800.0 PL=0
MOVL C01549 V=800.0 PL=0
MOVL C01550 V=800.0 PL=0
MOVL C01551 V=800.0 PL=0
MOVL C01552 V=800.0 PL=0
MOVL C01553 V=800.0 PL=0
MOVL C01554 V=800.0 PL=0
MOVL C01555 V=800.0 PL=0
MOVL C01556 V=800.0 PL=0
MOVL C01557 V=800.0 PL=0
MOVL C01558 V=800.0 PL=0
MOVL C01559 V=800.0 PL=0
MOVL C01560 V=800.0 PL=0
MOVL C01561 V=800.0 PL=0
MOVL C01562 V=800.0 PL=0
MOVL C01563 V=800.0 PL=0
MOVL C01564 V=800.0 PL=0
MOVL C01565 V=800.0 PL=0
MOVL C01566 V=800.0 PL=0
MOVL C01567 V=800.0 PL=0
MOVL C01568 V=800.0 PL=0
MOVL C01569 V=800.0 PL=0
MOVL C01570 V=800.0 PL=0
MOVL C01571 V=800.0 PL=0
MOVL C01572 V=800.0 PL=0
MOVL C01573 V=800.0 PL=0
MOVL C01574 V=800.0 PL=0
MOVL C01575 V=800.0 PL=0
MOVL C01576 V=800.0 PL=0
MOVL C01577 V=800.0 PL=0
MOVL C01578 V=800.0 PL=0
MOVL C01579 V=800.0 PL=0
MOVL C01580 V=800.0 PL=0
MOVL C01581 V=800.0 PL=0
MOVL C01582 V=800.0 PL=0
MOVL C01583 V=800.0 PL=0
MOVL C01584 V=800.0 PL=0
MOVL C01585 V=800.0 PL=0
MOVL C01586 V=800.0 PL=0
MOVL C01587 V=800.0 PL=0
MOVL C01588 V=800.0 PL=0
MOVL C01589 V=800.0 PL=0
MOVL C01590 V=800.0 PL=0
MOVL C01591 V=800.0 PL=0
MOVL C01592 V=800.0 PL=0
MOVL C01593 V=800.0 PL=0
MOVL C01594 V=800.0 PL=0
MOVL C01595 V=800.0 PL=0
MOVL C01596 V=800.0 PL=0
MOVL C01597 V=800.0 PL=0
MOVL C01598 V=800.0 PL=0
MOVL C01599 V=800.0 PL=0
MOVL C01600 V=800.0 PL=0
MOVL C01601 V=800.0 PL=0
MOVL C01602 V=800.0 PL=0
MOVL C01603 V=800.0 PL=0
MOVL C01604 V=800.0 PL=0
MOVL C01605 V=800.0 PL=0
MOVL C01606 V=800.0 PL=0
MOVL C01607 V=800.0 PL=0
MOVL C01608 V=800.0 PL=0
MOVL C01609 V=800.0 PL=0
MOVL C01610 V=800.0 PL=0
MOVL C01611 V=800.0 PL=0
MOVL C01612 V=800.0 PL=0
MOVL C01613 V=800.0 PL=0
MOVL C01614 V=800.0 PL=0
MOVL C01615 V=800.0 PL=0
MOVL C01616 V=800.0 PL=0
MOVL C01617 V=800.0 PL=0
MOVL C01618 V=800.0 PL=0
MOVL C01619 V=800.0 PL=0
MOVL C01620 V=800.0 PL=0
MOVL C01621 V=800.0 PL=0
MOVL C01622 V=800.0 PL=0
MOVL C01623 V=800.0 PL=0
MOVL C01624 V=800.0 PL=0
MOVL C01625 V=800.0 PL=0
MOVL C01626 V=800.0 PL=0
MOVL C01627 V=800.0 PL=0
MOVL C01628 V=800.0 PL=0
MOVL C01629 V=800.0 PL=0
MOVL C01630 V=800.0 PL=0
MOVL C01631 V=800.0 PL=0
MOVL C01632 V=800.0 PL=0
MOVL C01633 V=800.0 PL=0
MOVL C01634 V=800.0 PL=0
MOVL C01635 V=800.0 PL=0
MOVL C01636 V=800.0 PL=0
MOVL C01637 V=800.0 PL=0
MOVL C01638 V=800.0 PL=0
MOVL C01639 V=800.0 PL=0
MOVL C01640 V=800.0 PL=0
MOVL C01641 V=800.0 PL=0
MOVL C01642 V=800.0 PL=0
MOVL C01643 V=800.0 PL=0
MOVL C01644 V=800.0 PL=0
MOVL C01645 V=800.0 PL=0
MOVL C01646 V=800.0 PL=0
MOVL C01647 V=800.0 PL=0
MOVL C01648 V=800.0 PL=0
MOVL C01649 V=800.0 PL=0
MOVL C01650 V=800.0 PL=0
MOVL C01651 V=800.0 PL=0
MOVL C01652 V=800.0 PL=0
MOVL C01653 V=800.0 PL=0
MOVL C01654 V=800.0 PL=0
MOVL C01655 V=800.0 PL=0
MOVL C01656 V=800.0 PL=0
MOVL C01657 V=800.0 PL=0
MOVL C01658 V=800.0 PL=0
MOVL C01659 V=800.0 PL=0
MOVL C01660 V=800.0 PL=0
MOVL C01661 V=800.0 PL=0
MOVL C01662 V=800.0 PL=0
MOVL C01663 V=800.0 PL=0
MOVL C01664 V=800.0 PL=0
MOVL C01665 V=800.0 PL=0
MOVL C01666 V=800.0 PL=0
MOVL C01667 V=800.0 PL=0
MOVL C01668 V=800.0 PL=0
MOVL C01669 V=800.0 PL=0
MOVL C01670 V=800.0 PL=0
MOVL C01671 V=800.0 PL=0
MOVL C01672 V=800.0 PL=0
MOVL C01673 V=800.0 PL=0
MOVL C01674 V=800.0 PL=0
MOVL C01675 V=800.0 PL=0
MOVL C01676 V=800.0 PL=0
MOVL C01677 V=800.0 PL=0
MOVL C01678 V=800.0 PL=0
MOVL C01679 V=800.0 PL=0
MOVL C01680 V=800.0 PL=0
MOVL C01681 V=800.0 PL=0
MOVL C01682 V=800.0 PL=0
MOVL C01683 V=800.0 PL=0
MOVL C01684 V=800.0 PL=0
MOVL C01685 V=800.0 PL=0
MOVL C01686 V=800.0 PL=0
MOVL C01687 V=800.0 PL=0
MOVL C01688 V=800.0 PL=0
MOVL C01689 V=800.0 PL=0
MOVL C01690 V=800.0 PL=0
MOVL C01691 V=800.0 PL=0
MOVL C01692 V=800.0 PL=0
MOVL C01693 V=800.0 PL=0
MOVL C01694 V=800.0 PL=0
MOVL C01695 V=800.0 PL=0
MOVL C01696 V=800.0 PL=0
MOVL C01697 V=800.0 PL=0
MOVL C01698 V=800.0 PL=0
MOVL C01699 V=800.0 PL=0
MOVL C01700 V=800.0 PL=0
MOVL C01701 V=800.0 PL=0
MOVL C01702 V=800.0 PL=0
MOVL C01703 V=800.0 PL=0
MOVL C01704 V=800.0 PL=0
MOVL C01705 V=800.0 PL=0
MOVL C01706 V=800.0 PL=0
MOVL C01707 V=800.0 PL=0
MOVL C01708 V=800.0 PL=0
MOVL C01709 V=800.0 PL=0
MOVL C01710 V=800.0 PL=0
MOVL C01711 V=800.0 PL=0
MOVL C01712 V=800.0 PL=0
MOVL C01713 V=800.0 PL=0
MOVL C01714 V=800.0 PL=0
MOVL C01715 V=800.0 PL=0
MOVL C01716 V=800.0 PL=0
MOVL C01717 V=800.0 PL=0
MOVL C01718 V=800.0 PL=0
MOVL C01719 V=800.0 PL=0
MOVL C01720 V=800.0 PL=0
MOVL C01721 V=800.0 PL=0
MOVL C01722 V=800.0 PL=0
MOVL C01723 V=800.0 PL=0
MOVL C01724 V=800.0 PL=0
MOVL C01725 V=800.0 PL=0
MOVL C01726 V=800.0 PL=0
MOVL C01727 V=800.0 PL=0
MOVL C01728 V=800.0 PL=0
MOVL C01729 V=800.0 PL=0
MOVL C01730 V=800.0 PL=0
MOVL C01731 V=800.0 PL=0
MOVL C01732 V=800.0 PL=0
MOVL C01733 V=800.0 PL=0
MOVL C01734 V=800.0 PL=0
MOVL C01735 V=800.0 PL=0
MOVL C01736 V=800.0 PL=0
MOVL C01737 V=800.0 PL=0
MOVL C01738 V=800.0 PL=0
MOVL C01739 V=800.0 PL=0
MOVL C01740 V=800.0 PL=0
MOVL C01741 V=800.0 PL=0
MOVL C01742 V=800.0 PL=0
MOVL C01743 V=800.0 PL=0
MOVL C01744 V=800.0 PL=0
MOVL C01745 V=800.0 PL=0
MOVL C01746 V=800.0 PL=0
MOVL C01747 V=800.0 PL=0
MOVL C01748 V=800.0 PL=0
MOVL C01749 V=800.0 PL=0
MOVL C01750 V=800.0 PL=0
MOVL C01751 V=800.0 PL=0
MOVL C01752 V=800.0 PL=0
MOVL C01753 V=800.0 PL=0
MOVL C01754 V=800.0 PL=0
MOVL C01755 V=800.0 PL=0
MOVL C01756 V=800.0 PL=0
MOVL C01757 V=800.0 PL=0
MOVL C01758 V=800.0 PL=0
MOVL C01759 V=800.0 PL=0
MOVL C01760 V=800.0 PL=0
MOVL C01761 V=800.0 PL=0
MOVL C01762 V=800.0 PL=0
MOVL C01763 V=800.0 PL=0
MOVL C01764 V=800.0 PL=0
MOVL C01765 V=800.0 PL=0
MOVL C01766 V=800.0 PL=0
MOVL C01767 V=800.0 PL=0
MOVL C01768 V=800.0 PL=0
MOVL C01769 V=800.0 PL=0
MOVL C01770 V=800.0 PL=0
MOVL C01771 V=800.0 PL=0
MOVL C01772 V=800.0 PL=0
MOVL C01773 V=800.0 PL=0
MOVL C01774 V=800.0 PL=0
MOVL C01775 V=800.0 PL=0
MOVL C01776 V=800.0 PL=0
MOVL C01777 V=800.0 PL=0
MOVL C01778 V=800.0 PL=0
MOVL C01779 V=800.0 PL=0
MOVL C01780 V=800.0 PL=0
MOVL C01781 V=800.0 PL=0
MOVL C01782 V=800.0 PL=0
MOVL C01783 V=800.0 PL=0
MOVL C01784 V=800.0 PL=0
MOVL C01785 V=800.0 PL=0
MOVL C01786 V=800.0 PL=0
MOVL C01787 V=800.0 PL=0
MOVL C01788 V=800.0 PL=0
MOVL C01789 V=800.0 PL=0
MOVL C01790 V=800.0 PL=0
MOVL C01791 V=800.0 PL=0
MOVL C01792 V=800.0 PL=0
MOVL C01793 V=800.0 PL=0
MOVL C01794 V=800.0 PL=0
MOVL C01795 V=800.0 PL=0
MOVL C01796 V=800.0 PL=0
MOVL C01797 V=800.0 PL=0
MOVL C01798 V=800.0 PL=0
MOVL C01799 V=800.0 PL=0
MOVL C01800 V=800.0 PL=0
MOVL C01801 V=800.0 PL=0
MOVL C01802 V=800.0 PL=0
MOVL C01803 V=800.0 PL=0
MOVL C01804 V=800.0 PL=0
MOVL C01805 V=800.0 PL=0
MOVL C01806 V=800.0 PL=0
MOVL C01807 V=800.0 PL=0
MOVL C01808 V=800.0 PL=0
MOVL C01809 V=800.0 PL=0
MOVL C01810 V=800.0 PL=0
MOVL C01811 V=800.0 PL=0
MOVL C01812 V=800.0 PL=0
MOVL C01813 V=800.0 PL=0
MOVL C01814 V=800.0 PL=0
MOVL C01815 V=800.0 PL=0
MOVL C01816 V=800.0 PL=0
MOVL C01817 V=800.0 PL=0
MOVL C01818 V=800.0 PL=0
MOVL C01819 V=800.0 PL=0
MOVL C01820 V=800.0 PL=0
MOVL C01821 V=800.0 PL=0
MOVL C01822 V=800.0 PL=0
MOVL C01823 V=800.0 PL=0
MOVL C01824 V=800.0 PL=0
MOVL C01825 V=800.0 PL=0
MOVL C01826 V=800.0 PL=0
MOVL C01827 V=800.0 PL=0
MOVL C01828 V=800.0 PL=0
MOVL C01829 V=800.0 PL=0
MOVL C01830 V=800.0 PL=0
MOVL C01831 V=800.0 PL=0
MOVL C01832 V=800.0 PL=0
MOVL C01833 V=800.0 PL=0
MOVL C01834 V=800.0 PL=0
MOVL C01835 V=800.0 PL=0
MOVL C01836 V=800.0 PL=0
MOVL C01837 V=800.0 PL=0
MOVL C01838 V=800.0 PL=0
MOVL C01839 V=800.0 PL=0
MOVL C01840 V=800.0 PL=0
MOVL C01841 V=800.0 PL=0
MOVL C01842 V=800.0 PL=0
MOVL C01843 V=800.0 PL=0
MOVL C01844 V=800.0 PL=0
MOVL C01845 V=800.0 PL=0
MOVL C01846 V=800.0 PL=0
MOVL C01847 V=800.0 PL=0
MOVL C01848 V=800.0 PL=0
MOVL C01849 V=800.0 PL=0
MOVL C01850 V=800.0 PL=0
MOVL C01851 V=800.0 PL=0
MOVL C01852 V=800.0 PL=0
MOVL C01853 V=800.0 PL=0
MOVL C01854 V=800.0 PL=0
MOVL C01855 V=800.0 PL=0
MOVL C01856 V=800.0 PL=0
MOVL C01857 V=800.0 PL=0
MOVL C01858 V=800.0 PL=0
MOVL C01859 V=800.0 PL=0
MOVL C01860 V=800.0 PL=0
MOVL C01861 V=800.0 PL=0
MOVL C01862 V=800.0 PL=0
MOVL C01863 V=800.0 PL=0
MOVL C01864 V=800.0 PL=0
MOVL C01865 V=800.0 PL=0
MOVL C01866 V=800.0 PL=0
MOVL C01867 V=800.0 PL=0
MOVL C01868 V=800.0 PL=0
MOVL C01869 V=800.0 PL=0
MOVL C01870 V=800.0 PL=0
MOVL C01871 V=800.0 PL=0
MOVL C01872 V=800.0 PL=0
MOVL C01873 V=800.0 PL=0
MOVL C01874 V=800.0 PL=0
MOVL C01875 V=800.0 PL=0
MOVL C01876 V=800.0 PL=0
MOVL C01877 V=800.0 PL=0
MOVL C01878 V=800.0 PL=0
MOVL C01879 V=800.0 PL=0
MOVL C01880 V=800.0 PL=0
MOVL C01881 V=800.0 PL=0
MOVL C01882 V=800.0 PL=0
MOVL C01883 V=800.0 PL=0
MOVL C01884 V=800.0 PL=0
MOVL C01885 V=800.0 PL=0
MOVL C01886 V=800.0 PL=0
MOVL C01887 V=800.0 PL=0
MOVL C01888 V=800.0 PL=0
MOVL C01889 V=800.0 PL=0
MOVL C01890 V=800.0 PL=0
MOVL C01891 V=800.0 PL=0
MOVL C01892 V=800.0 PL=0
MOVL C01893 V=800.0 PL=0
MOVL C01894 V=800.0 PL=0
MOVL C01895 V=800.0 PL=0
MOVL C01896 V=800.0 PL=0
MOVL C01897 V=800.0 PL=0
MOVL C01898 V=800.0 PL=0
MOVL C01899 V=800.0 PL=0
MOVL C01900 V=800.0 PL=0
MOVL C01901 V=800.0 PL=0
MOVL C01902 V=800.0 PL=0
MOVL C01903 V=800.0 PL=0
MOVL C01904 V=800.0 PL=0
MOVL C01905 V=800.0 PL=0
MOVL C01906 V=800.0 PL=0
MOVL C01907 V=800.0 PL=0
MOVL C01908 V=800.0 PL=0
MOVL C01909 V=800.0 PL=0
MOVL C01910 V=800.0 PL=0
MOVL C01911 V=800.0 PL=0
MOVL C01912 V=800.0 PL=0
MOVL C01913 V=800.0 PL=0
MOVL C01914 V=800.0 PL=0
MOVL C01915 V=800.0 PL=0
MOVL C01916 V=800.0 PL=0
MOVL C01917 V=800.0 PL=0
MOVL C01918 V=800.0 PL=0
MOVL C01919 V=800.0 PL=0
MOVL C01920 V=800.0 PL=0
MOVL C01921 V=800.0 PL=0
MOVL C01922 V=800.0 PL=0
MOVL C01923 V=800.0 PL=0
MOVL C01924 V=800.0 PL=0
MOVL C01925 V=800.0 PL=0
MOVL C01926 V=800.0 PL=0
MOVL C01927 V=800.0 PL=0
MOVL C01928 V=800.0 PL=0
MOVL C01929 V=800.0 PL=0
MOVL C01930 V=800.0 PL=0
MOVL C01931 V=800.0 PL=0
MOVL C01932 V=800.0 PL=0
MOVL C01933 V=800.0 PL=0
MOVL C01934 V=800.0 PL=0
MOVL C01935 V=800.0 PL=0
MOVL C01936 V=800.0 PL=0
MOVL C01937 V=800.0 PL=0
MOVL C01938 V=800.0 PL=0
MOVL C01939 V=800.0 PL=0
MOVL C01940 V=800.0 PL=0
MOVL C01941 V=800.0 PL=0
MOVL C01942 V=800.0 PL=0
MOVL C01943 V=800.0 PL=0
MOVL C01944 V=800.0 PL=0
MOVL C01945 V=800.0 PL=0
MOVL C01946 V=800.0 PL=0
MOVL C01947 V=800.0 PL=0
MOVL C01948 V=800.0 PL=0
MOVL C01949 V=800.0 PL=0
MOVL C01950 V=800.0 PL=0
MOVL C01951 V=800.0 PL=0
MOVL C01952 V=800.0 PL=0
MOVL C01953 V=800.0 PL=0
MOVL C01954 V=800.0 PL=0
MOVL C01955 V=800.0 PL=0
MOVL C01956 V=800.0 PL=0
MOVL C01957 V=800.0 PL=0
MOVL C01958 V=800.0 PL=0
MOVL C01959 V=800.0 PL=0
MOVL C01960 V=800.0 PL=0
MOVL C01961 V=800.0 PL=0
MOVL C01962 V=800.0 PL=0
MOVL C01963 V=800.0 PL=0
MOVL C01964 V=800.0 PL=0
MOVL C01965 V=800.0 PL=0
MOVL C01966 V=800.0 PL=0
MOVL C01967 V=800.0 PL=0
MOVL C01968 V=800.0 PL=0
MOVL C01969 V=800.0 PL=0
MOVL C01970 V=800.0 PL=0
MOVL C01971 V=800.0 PL=0
MOVL C01972 V=800.0 PL=0
MOVL C01973 V=800.0 PL=0
MOVL C01974 V=800.0 PL=0
MOVL C01975 V=800.0 PL=0
MOVL C01976 V=800.0 PL=0
MOVL C01977 V=800.0 PL=0
MOVL C01978 V=800.0 PL=0
MOVL C01979 V=800.0 PL=0
MOVL C01980 V=800.0 PL=0
MOVL C01981 V=800.0 PL=0
MOVL C01982 V=800.0 PL=0
MOVL C01983 V=800.0 PL=0
MOVL C01984 V=800.0 PL=0
MOVL C01985 V=800.0 PL=0
MOVL C01986 V=800.0 PL=0
MOVL C01987 V=800.0 PL=0
MOVL C01988 V=800.0 PL=0
MOVL C01989 V=800.0 PL=0
MOVL C01990 V=800.0 PL=0
MOVL C01991 V=800.0 PL=0
MOVL C01992 V=800.0 PL=0
MOVL C01993 V=800.0 PL=0
MOVL C01994 V=800.0 PL=0
MOVL C01995 V=800.0 PL=0
MOVL C01996 V=800.0 PL=0
MOVL C01997 V=800.0 PL=0
MOVL C01998 V=800.0 PL=0
MOVL C01999 V=800.0 PL=0
MOVL C02000 V=800.0 PL=0
MOVL C02001 V=800.0 PL=0
MOVL C02002 V=800.0 PL=0
MOVL C02003 V=800.0 PL=0
MOVL C02004 V=800.0 PL=0
MOVL C02005 V=800.0 PL=0
MOVL C02006 V=800.0 PL=0
MOVL C02007 V=800.0 PL=0
MOVL C02008 V=800.0 PL=0
MOVL C02009 V=800.0 PL=0
MOVL C02010 V=800.0 PL=0
MOVL C02011 V=800.0 PL=0
MOVL C02012 V=800.0 PL=0
MOVL C02013 V=800.0 PL=0
MOVL C02014 V=800.0 PL=0
MOVL C02015 V=800.0 PL=0
MOVL C02016 V=800.0 PL=0
MOVL C02017 V=800.0 PL=0
MOVL C02018 V=800.0 PL=0
MOVL C02019 V=800.0 PL=0
MOVL C02020 V=800.0 PL=0
MOVL C02021 V=800.0 PL=0
MOVL C02022 V=800.0 PL=0
MOVL C02023 V=800.0 PL=0
MOVL C02024 V=800.0 PL=0
